LIN {X 0.001,Y -175.729,Z 1561.412,A 0.000,B 0.000,C 90.000,E1 254.212} C_DIS
LIN {X -0.003,Y -171.914,Z 1561.384,A 0.000,B 0.000,C 90.000,E1 249.082} C_DIS
LIN {X -0.028,Y -171.279,Z 1561.379,A 0.000,B 0.000,C 90.000,E1 248.230} C_DIS
LIN {X 0.018,Y -167.547,Z 1561.355,A 0.000,B 0.000,C 90.000,E1 243.896} C_DIS
LIN {X 0.032,Y -166.166,Z 1561.345,A 0.000,B 0.000,C 90.000,E1 242.153} C_DIS
LIN {X 0.022,Y -162.940,Z 1561.326,A 0.000,B 0.000,C 90.000,E1 238.663} C_DIS
LIN {X -0.001,Y -161.611,Z 1561.316,A 0.000,B 0.000,C 90.000,E1 236.914} C_DIS
LIN {X -0.025,Y -159.137,Z 1561.302,A 0.000,B 0.000,C 90.000,E1 234.276} C_DIS
LIN {X -0.014,Y -155.659,Z 1561.277,A 0.000,B 0.000,C 90.000,E1 229.828} C_DIS
LIN {X 0.038,Y -151.928,Z 1561.252,A 0.000,B 0.000,C 90.000,E1 225.324} C_DIS
LIN {X 0.053,Y -150.165,Z 1561.237,A 0.000,B 0.000,C 90.000,E1 222.609} C_DIS
LIN {X -0.027,Y -146.943,Z 1561.212,A 0.000,B 0.000,C 90.000,E1 218.096} C_DIS
LIN {X 0.079,Y -145.531,Z 1561.196,A 0.000,B 0.000,C 90.000,E1 215.311} C_DIS
LIN {X 0.000,Y -142.929,Z 1561.171,A 0.000,B 0.000,C 90.000,E1 210.747} C_DIS
LIN {X 0.000,Y -141.552,Z 1561.150,A 0.000,B 0.000,C 90.000,E1 207.052} C_DIS
LIN {X -0.011,Y -139.406,Z 1561.114,A 0.000,B 0.000,C 90.000,E1 200.556} C_DIS
LIN {X 0.042,Y -139.125,Z 1561.104,A 0.000,B 0.000,C 90.000,E1 198.671} C_DIS
LIN {X -0.063,Y -138.351,Z 1561.057,A 0.000,B 0.000,C 90.000,E1 190.310} C_DIS
LIN {X 0.064,Y -139.501,Z 1561.005,A 0.000,B 0.000,C 90.000,E1 180.917} C_DIS
LIN {X 0.005,Y -141.127,Z 1560.974,A 0.000,B 0.000,C 90.000,E1 175.355} C_DIS
LIN {X -0.041,Y -142.507,Z 1560.959,A 0.000,B 0.000,C 90.000,E1 172.591} C_DIS
LIN {X 0.045,Y -144.765,Z 1560.933,A 0.000,B 0.000,C 90.000,E1 167.937} C_DIS
LIN {X -0.005,Y -147.378,Z 1560.913,A 0.000,B 0.000,C 90.000,E1 164.283} C_DIS
LIN {X 0.058,Y -150.706,Z 1560.887,A 0.000,B 0.000,C 90.000,E1 159.699} C_DIS
LIN {X -0.001,Y -154.187,Z 1560.867,A 0.000,B 0.000,C 90.000,E1 156.102} C_DIS
LIN {X 0.068,Y -157.624,Z 1560.847,A 0.000,B 0.000,C 90.000,E1 152.487} C_DIS
LIN {X 0.017,Y -161.879,Z 1560.828,A 0.000,B 0.000,C 90.000,E1 148.948} C_DIS
LIN {X -0.011,Y -166.070,Z 1560.808,A 0.000,B 0.000,C 90.000,E1 145.435} C_DIS
LIN {X -0.010,Y -171.076,Z 1560.789,A 0.000,B 0.000,C 90.000,E1 141.949} C_DIS
LIN {X 0.045,Y -175.949,Z 1560.769,A 0.000,B 0.000,C 90.000,E1 138.485} C_DIS
LIN {X -0.095,Y -180.192,Z 1560.755,A 0.000,B 0.000,C 90.000,E1 135.972} C_DIS
LIN {X 0.010,Y -185.607,Z 1560.736,A 0.000,B 0.000,C 90.000,E1 132.567} C_DIS
LIN {X -0.078,Y -190.201,Z 1560.723,A 0.000,B 0.000,C 90.000,E1 130.092} C_DIS
LIN {X -0.034,Y -197.529,Z 1560.700,A 0.000,B 0.000,C 90.000,E1 125.964} C_DIS
LIN {X 0.007,Y -200.796,Z 1560.691,A 0.000,B 0.000,C 90.000,E1 124.326} C_DIS
LIN {X 0.030,Y -203.630,Z 1560.682,A 0.000,B 0.000,C 90.000,E1 122.704} C_DIS
LIN {X 0.011,Y -319.680,Z 1560.682,A 0.000,B 0.000,C 90.000,E1 122.704} C_DIS
LIN {X -0.131,Y -322.536,Z 1560.681,A 0.000,B 0.000,C 90.000,E1 122.673} C_DIS
LIN {X -0.011,Y -326.250,Z 1560.680,A 0.000,B 0.000,C 90.000,E1 122.467} C_DIS
LIN {X -0.066,Y -328.541,Z 1560.679,A 0.000,B 0.000,C 90.000,E1 122.291} C_DIS
LIN {X -0.102,Y -331.721,Z 1560.677,A 0.000,B 0.000,C 90.000,E1 121.926} C_DIS
LIN {X 0.040,Y -333.633,Z 1560.676,A 0.000,B 0.000,C 90.000,E1 121.592} C_DIS
LIN {X 0.184,Y -335.119,Z 1560.674,A 0.000,B 0.000,C 90.000,E1 121.258} C_DIS
LIN {X -0.201,Y -347.889,Z 1560.657,A 0.000,B 0.000,C 90.000,E1 118.231} C_DIS
LIN {X 0.062,Y -360.849,Z 1560.641,A 0.000,B 0.000,C 90.000,E1 115.463} C_DIS
LIN {X -0.104,Y -375.345,Z 1560.627,A 0.000,B 0.000,C 90.000,E1 112.823} C_DIS
LIN {X 0.048,Y -389.617,Z 1560.614,A 0.000,B 0.000,C 90.000,E1 110.482} C_DIS
LIN {X -0.079,Y -405.297,Z 1560.601,A 0.000,B 0.000,C 90.000,E1 108.236} C_DIS
LIN {X -0.073,Y -422.494,Z 1560.589,A 0.000,B 0.000,C 90.000,E1 106.024} C_DIS
LIN {X -0.171,Y -441.327,Z 1560.577,A 0.000,B 0.000,C 90.000,E1 103.883} C_DIS
LIN {X 0.024,Y -461.282,Z 1560.566,A 0.000,B 0.000,C 90.000,E1 101.827} C_DIS
LIN {X 0.129,Y -484.372,Z 1560.554,A 0.000,B 0.000,C 90.000,E1 99.726} C_DIS
LIN {X -0.075,Y -492.225,Z 1560.551,A 0.000,B 0.000,C 90.000,E1 99.095} C_DIS
LIN {X 0.121,Y -494.492,Z 1560.549,A 0.000,B 0.000,C 90.000,E1 98.859} C_DIS
LIN {X -0.171,Y -496.210,Z 1560.548,A 0.000,B 0.000,C 90.000,E1 98.681} C_DIS
LIN {X 0.161,Y -497.718,Z 1560.547,A 0.000,B 0.000,C 90.000,E1 98.398} C_DIS
LIN {X 0.076,Y -498.838,Z 1560.545,A 0.000,B 0.000,C 90.000,E1 98.163} C_DIS
LIN {X -0.149,Y -500.153,Z 1560.543,A 0.000,B 0.000,C 90.000,E1 97.701} C_DIS
LIN {X 0.129,Y -500.420,Z 1560.540,A 0.000,B 0.000,C 90.000,E1 97.182} C_DIS
LIN {X -0.082,Y -499.687,Z 1560.537,A 0.000,B 0.000,C 90.000,E1 96.720} C_DIS
LIN {X 0.206,Y -497.830,Z 1560.535,A 0.000,B 0.000,C 90.000,E1 96.201} C_DIS
LIN {X -0.007,Y -494.661,Z 1560.532,A 0.000,B 0.000,C 90.000,E1 95.739} C_DIS
LIN {X 0.042,Y -478.703,Z 1560.518,A 0.000,B 0.000,C 90.000,E1 93.269} C_DIS
LIN {X -0.049,Y -468.865,Z 1560.510,A 0.000,B 0.000,C 90.000,E1 91.776} C_DIS
LIN {X 0.123,Y -458.506,Z 1560.501,A 0.000,B 0.000,C 90.000,E1 90.229} C_DIS
LIN {X -0.099,Y -449.397,Z 1560.494,A 0.000,B 0.000,C 90.000,E1 88.969} C_DIS
LIN {X 0.015,Y -439.937,Z 1560.487,A 0.000,B 0.000,C 90.000,E1 87.650} C_DIS
LIN {X 0.131,Y -428.188,Z 1560.478,A 0.000,B 0.000,C 90.000,E1 86.045} C_DIS
LIN {X 0.189,Y -414.521,Z 1560.468,A 0.000,B 0.000,C 90.000,E1 84.147} C_DIS
LIN {X -0.172,Y -395.787,Z 1560.452,A 0.000,B 0.000,C 90.000,E1 81.432} C_DIS
LIN {X -0.071,Y -376.486,Z 1560.435,A 0.000,B 0.000,C 90.000,E1 78.285} C_DIS
LIN {X -0.026,Y -361.558,Z 1560.420,A 0.000,B 0.000,C 90.000,E1 75.644} C_DIS
LIN {X -0.138,Y -348.671,Z 1560.407,A 0.000,B 0.000,C 90.000,E1 73.268} C_DIS
LIN {X 0.078,Y -335.994,Z 1560.393,A 0.000,B 0.000,C 90.000,E1 70.786} C_DIS
LIN {X 0.056,Y -322.338,Z 1560.378,A 0.000,B 0.000,C 90.000,E1 67.975} C_DIS
LIN {X 0.048,Y -312.282,Z 1560.365,A 0.000,B 0.000,C 90.000,E1 65.741} C_DIS
LIN {X 0.103,Y -300.822,Z 1560.351,A 0.000,B 0.000,C 90.000,E1 63.127} C_DIS
LIN {X -0.098,Y -290.975,Z 1560.338,A 0.000,B 0.000,C 90.000,E1 60.845} C_DIS
LIN {X 0.028,Y -281.124,Z 1560.325,A 0.000,B 0.000,C 90.000,E1 58.456} C_DIS
LIN {X -0.135,Y -268.850,Z 1560.307,A 0.000,B 0.000,C 90.000,E1 55.388} C_DIS
LIN {X -0.076,Y -258.197,Z 1560.292,A 0.000,B 0.000,C 90.000,E1 52.557} C_DIS
LIN {X -0.003,Y -246.691,Z 1560.274,A 0.000,B 0.000,C 90.000,E1 49.299} C_DIS
LIN {X 0.047,Y -235.998,Z 1560.255,A 0.000,B 0.000,C 90.000,E1 45.972} C_DIS
LIN {X 0.018,Y -227.267,Z 1560.239,A 0.000,B 0.000,C 90.000,E1 42.975} C_DIS
LIN {X -0.017,Y -219.351,Z 1560.222,A 0.000,B 0.000,C 90.000,E1 39.930} C_DIS
LIN {X 0.120,Y -212.173,Z 1560.205,A 0.000,B 0.000,C 90.000,E1 36.790} C_DIS
LIN {X 0.045,Y -205.796,Z 1560.187,A 0.000,B 0.000,C 90.000,E1 33.658} C_DIS
LIN {X 0.048,Y -200.192,Z 1560.169,A 0.000,B 0.000,C 90.000,E1 30.463} C_DIS
LIN {X -0.046,Y -195.357,Z 1560.151,A 0.000,B 0.000,C 90.000,E1 27.257} C_DIS
LIN {X 0.003,Y -190.249,Z 1560.129,A 0.000,B 0.000,C 90.000,E1 23.153} C_DIS
LIN {X -0.042,Y -186.042,Z 1560.106,A 0.000,B 0.000,C 90.000,E1 19.033} C_DIS
LIN {X 0.003,Y -181.949,Z 1560.078,A 0.000,B 0.000,C 90.000,E1 14.008} C_DIS
LIN {X 0.022,Y -179.288,Z 1560.054,A 0.000,B 0.000,C 90.000,E1 9.792} C_DIS
LIN {X 0.074,Y -176.632,Z 1560.021,A 0.000,B 0.000,C 90.000,E1 3.841} C_DIS
LIN {X 0.076,Y -175.789,Z 1559.974,A 0.000,B 0.000,C 90.000,E1 355.241} C_DIS
LIN {X 0.028,Y -177.969,Z 1559.931,A 0.000,B 0.000,C 90.000,E1 347.589} C_DIS
LIN {X -0.093,Y -181.069,Z 1559.903,A 0.000,B 0.000,C 90.000,E1 342.543} C_DIS
LIN {X 0.078,Y -184.847,Z 1559.880,A 0.000,B 0.000,C 90.000,E1 338.284} C_DIS
LIN {X -0.043,Y -189.476,Z 1559.856,A 0.000,B 0.000,C 90.000,E1 334.152} C_DIS
LIN {X -0.028,Y -193.917,Z 1559.838,A 0.000,B 0.000,C 90.000,E1 330.845} C_DIS
LIN {X -0.049,Y -198.981,Z 1559.820,A 0.000,B 0.000,C 90.000,E1 327.582} C_DIS
LIN {X 0.046,Y -204.824,Z 1559.802,A 0.000,B 0.000,C 90.000,E1 324.322} C_DIS
LIN {X -0.094,Y -211.403,Z 1559.784,A 0.000,B 0.000,C 90.000,E1 321.170} C_DIS
LIN {X 0.001,Y -218.920,Z 1559.767,A 0.000,B 0.000,C 90.000,E1 318.000} C_DIS
LIN {X 0.062,Y -228.250,Z 1559.747,A 0.000,B 0.000,C 90.000,E1 314.514} C_DIS
LIN {X -0.049,Y -237.564,Z 1559.731,A 0.000,B 0.000,C 90.000,E1 311.515} C_DIS
LIN {X -0.017,Y -244.136,Z 1559.720,A 0.000,B 0.000,C 90.000,E1 309.644} C_DIS
LIN {X -0.035,Y -250.151,Z 1559.712,A 0.000,B 0.000,C 90.000,E1 308.177} C_DIS
LIN {X -0.103,Y -258.667,Z 1559.702,A 0.000,B 0.000,C 90.000,E1 306.377} C_DIS
LIN {X 0.121,Y -266.282,Z 1559.694,A 0.000,B 0.000,C 90.000,E1 304.898} C_DIS
LIN {X -0.001,Y -276.782,Z 1559.684,A 0.000,B 0.000,C 90.000,E1 303.166} C_DIS
LIN {X 0.063,Y -297.972,Z 1559.667,A 0.000,B 0.000,C 90.000,E1 300.079} C_DIS
LIN {X 0.067,Y -315.483,Z 1559.654,A 0.000,B 0.000,C 90.000,E1 297.769} C_DIS
LIN {X 0.063,Y -330.718,Z 1559.644,A 0.000,B 0.000,C 90.000,E1 295.848} C_DIS
LIN {X -0.091,Y -346.011,Z 1559.633,A 0.000,B 0.000,C 90.000,E1 294.003} C_DIS
LIN {X 0.134,Y -366.686,Z 1559.620,A 0.000,B 0.000,C 90.000,E1 291.589} C_DIS
LIN {X 0.107,Y -379.285,Z 1559.612,A 0.000,B 0.000,C 90.000,E1 290.194} C_DIS
LIN {X 0.153,Y -389.278,Z 1559.606,A 0.000,B 0.000,C 90.000,E1 289.033} C_DIS
LIN {X 0.119,Y -396.170,Z 1559.601,A 0.000,B 0.000,C 90.000,E1 288.181} C_DIS
LIN {X 0.032,Y -402.390,Z 1559.596,A 0.000,B 0.000,C 90.000,E1 287.347} C_DIS
LIN {X 0.114,Y -407.864,Z 1559.592,A 0.000,B 0.000,C 90.000,E1 286.496} C_DIS
LIN {X -0.086,Y -411.083,Z 1559.589,A 0.000,B 0.000,C 90.000,E1 285.969} C_DIS
LIN {X -0.036,Y -415.144,Z 1559.584,A 0.000,B 0.000,C 90.000,E1 285.134} C_DIS
LIN {X 0.046,Y -418.481,Z 1559.579,A 0.000,B 0.000,C 90.000,E1 284.300} C_DIS
LIN {X -0.084,Y -420.231,Z 1559.576,A 0.000,B 0.000,C 90.000,E1 283.772} C_DIS
LIN {X -0.111,Y -421.582,Z 1559.573,A 0.000,B 0.000,C 90.000,E1 283.231} C_DIS
LIN {X 0.184,Y -422.530,Z 1559.570,A 0.000,B 0.000,C 90.000,E1 282.647} C_DIS
LIN {X 0.076,Y -422.973,Z 1559.567,A 0.000,B 0.000,C 90.000,E1 282.119} C_DIS
LIN {X -0.025,Y -422.940,Z 1559.564,A 0.000,B 0.000,C 90.000,E1 281.591} C_DIS
LIN {X -0.207,Y -422.407,Z 1559.561,A 0.000,B 0.000,C 90.000,E1 281.074} C_DIS
LIN {X 0.108,Y -421.297,Z 1559.558,A 0.000,B 0.000,C 90.000,E1 280.489} C_DIS
LIN {X 0.005,Y -419.589,Z 1559.555,A 0.000,B 0.000,C 90.000,E1 279.962} C_DIS
LIN {X -0.107,Y -417.240,Z 1559.552,A 0.000,B 0.000,C 90.000,E1 279.434} C_DIS
LIN {X 0.107,Y -414.174,Z 1559.549,A 0.000,B 0.000,C 90.000,E1 278.859} C_DIS
LIN {X -0.101,Y -410.312,Z 1559.546,A 0.000,B 0.000,C 90.000,E1 278.341} C_DIS
LIN {X 0.137,Y -405.638,Z 1559.543,A 0.000,B 0.000,C 90.000,E1 277.757} C_DIS
LIN {X -0.110,Y -400.056,Z 1559.540,A 0.000,B 0.000,C 90.000,E1 277.239} C_DIS
LIN {X -0.046,Y -394.108,Z 1559.537,A 0.000,B 0.000,C 90.000,E1 276.720} C_DIS
LIN {X -0.043,Y -387.993,Z 1559.535,A 0.000,B 0.000,C 90.000,E1 276.258} C_DIS
LIN {X -0.145,Y -381.773,Z 1559.532,A 0.000,B 0.000,C 90.000,E1 275.853} C_DIS
LIN {X -0.039,Y -375.314,Z 1559.530,A 0.000,B 0.000,C 90.000,E1 275.454} C_DIS
LIN {X 0.086,Y -365.730,Z 1559.527,A 0.000,B 0.000,C 90.000,E1 274.935} C_DIS
LIN {X 0.155,Y -355.917,Z 1559.525,A 0.000,B 0.000,C 90.000,E1 274.473} C_DIS
LIN {X -0.030,Y -340.256,Z 1559.521,A 0.000,B 0.000,C 90.000,E1 273.841} C_DIS
LIN {X 0.136,Y -327.066,Z 1559.519,A 0.000,B 0.000,C 90.000,E1 273.326} C_DIS
LIN {X -0.086,Y -316.982,Z 1559.517,A 0.000,B 0.000,C 90.000,E1 273.037} C_DIS
LIN {X -0.084,Y -306.535,Z 1559.515,A 0.000,B 0.000,C 90.000,E1 272.751} C_DIS
LIN {X 0.118,Y -295.128,Z 1559.514,A 0.000,B 0.000,C 90.000,E1 272.465} C_DIS
LIN {X 0.004,Y -282.361,Z 1559.513,A 0.000,B 0.000,C 90.000,E1 272.293} C_DIS
LIN {X 0.048,Y -267.759,Z 1559.512,A 0.000,B 0.000,C 90.000,E1 272.121} C_DIS
LIN {X -0.013,Y -258.424,Z 1559.511,A 0.000,B 0.000,C 90.000,E1 272.064} C_DIS
LIN {X 0.060,Y -246.056,Z 1559.511,A 0.000,B 0.000,C 90.000,E1 272.007} C_DIS
LIN {X 0.016,Y -181.260,Z 1559.511,A 0.000,B 0.000,C 90.000,E1 272.007} C_DIS
LIN {X -0.008,Y -181.581,Z 1559.502,A 0.000,B 0.000,C 90.000,E1 270.286} C_DIS
LIN {X -0.032,Y -180.898,Z 1559.474,A 0.000,B 0.000,C 90.000,E1 265.241} C_DIS
LIN {X -0.083,Y -180.212,Z 1559.464,A 0.000,B 0.000,C 90.000,E1 263.571} C_DIS
LIN {X 0.047,Y -179.032,Z 1559.445,A 0.000,B 0.000,C 90.000,E1 260.151} C_DIS
LIN {X -0.066,Y -178.688,Z 1559.441,A 0.000,B 0.000,C 90.000,E1 259.342} C_DIS
LIN {X 0.044,Y -175.738,Z 1559.412,A 0.000,B 0.000,C 90.000,E1 254.212} C_DIS
LIN {X 0.040,Y -171.922,Z 1559.384,A 0.000,B 0.000,C 90.000,E1 249.082} C_DIS
LIN {X 0.014,Y -171.294,Z 1559.379,A 0.000,B 0.000,C 90.000,E1 248.230} C_DIS
LIN {X 0.060,Y -167.558,Z 1559.355,A 0.000,B 0.000,C 90.000,E1 243.896} C_DIS
LIN {X 0.074,Y -166.181,Z 1559.345,A 0.000,B 0.000,C 90.000,E1 242.153} C_DIS
LIN {X 0.063,Y -162.952,Z 1559.326,A 0.000,B 0.000,C 90.000,E1 238.663} C_DIS
LIN {X 0.111,Y -160.859,Z 1559.311,A 0.000,B 0.000,C 90.000,E1 236.008} C_DIS
LIN {X 0.088,Y -157.635,Z 1559.292,A 0.000,B 0.000,C 90.000,E1 232.477} C_DIS
LIN {X 0.025,Y -155.672,Z 1559.277,A 0.000,B 0.000,C 90.000,E1 229.828} C_DIS
LIN {X 0.077,Y -151.940,Z 1559.252,A 0.000,B 0.000,C 90.000,E1 225.324} C_DIS
LIN {X 0.092,Y -150.176,Z 1559.237,A 0.000,B 0.000,C 90.000,E1 222.609} C_DIS
LIN {X 0.012,Y -146.952,Z 1559.212,A 0.000,B 0.000,C 90.000,E1 218.096} C_DIS
LIN {X -0.001,Y -145.540,Z 1559.196,A 0.000,B 0.000,C 90.000,E1 215.358} C_DIS
LIN {X 0.039,Y -142.936,Z 1559.171,A 0.000,B 0.000,C 90.000,E1 210.747} C_DIS
LIN {X -0.027,Y -141.559,Z 1559.150,A 0.000,B 0.000,C 90.000,E1 207.078} C_DIS
LIN {X 0.026,Y -139.408,Z 1559.114,A 0.000,B 0.000,C 90.000,E1 200.556} C_DIS
LIN {X -0.053,Y -139.129,Z 1559.104,A 0.000,B 0.000,C 90.000,E1 198.725} C_DIS
LIN {X -0.025,Y -138.350,Z 1559.057,A 0.000,B 0.000,C 90.000,E1 190.310} C_DIS
LIN {X -0.037,Y -139.499,Z 1559.005,A 0.000,B 0.000,C 90.000,E1 180.974} C_DIS
LIN {X 0.044,Y -141.121,Z 1558.974,A 0.000,B 0.000,C 90.000,E1 175.355} C_DIS
LIN {X -0.004,Y -142.500,Z 1558.959,A 0.000,B 0.000,C 90.000,E1 172.591} C_DIS
LIN {X -0.057,Y -144.756,Z 1558.933,A 0.000,B 0.000,C 90.000,E1 167.993} C_DIS
LIN {X 0.034,Y -147.366,Z 1558.913,A 0.000,B 0.000,C 90.000,E1 164.283} C_DIS
LIN {X -0.043,Y -150.693,Z 1558.887,A 0.000,B 0.000,C 90.000,E1 159.752} C_DIS
LIN {X 0.039,Y -154.173,Z 1558.867,A 0.000,B 0.000,C 90.000,E1 156.102} C_DIS
LIN {X -0.031,Y -157.607,Z 1558.847,A 0.000,B 0.000,C 90.000,E1 152.538} C_DIS
LIN {X 0.058,Y -161.860,Z 1558.828,A 0.000,B 0.000,C 90.000,E1 148.948} C_DIS
LIN {X -0.063,Y -166.051,Z 1558.808,A 0.000,B 0.000,C 90.000,E1 145.468} C_DIS
LIN {X -0.072,Y -171.055,Z 1558.789,A 0.000,B 0.000,C 90.000,E1 141.984} C_DIS
LIN {X -0.043,Y -175.927,Z 1558.770,A 0.000,B 0.000,C 90.000,E1 138.528} C_DIS
LIN {X -0.051,Y -180.166,Z 1558.755,A 0.000,B 0.000,C 90.000,E1 135.972} C_DIS
LIN {X -0.082,Y -185.583,Z 1558.737,A 0.000,B 0.000,C 90.000,E1 132.609} C_DIS
LIN {X -0.033,Y -190.174,Z 1558.723,A 0.000,B 0.000,C 90.000,E1 130.092} C_DIS
LIN {X 0.012,Y -197.502,Z 1558.700,A 0.000,B 0.000,C 90.000,E1 125.964} C_DIS
LIN {X 0.054,Y -200.772,Z 1558.691,A 0.000,B 0.000,C 90.000,E1 124.326} C_DIS
LIN {X -0.015,Y -203.565,Z 1558.682,A 0.000,B 0.000,C 90.000,E1 122.752} C_DIS
LIN {X -0.066,Y -319.571,Z 1558.682,A 0.000,B 0.000,C 90.000,E1 122.752} C_DIS
LIN {X 0.011,Y -323.866,Z 1558.681,A 0.000,B 0.000,C 90.000,E1 122.625} C_DIS
LIN {X 0.047,Y -327.091,Z 1558.680,A 0.000,B 0.000,C 90.000,E1 122.418} C_DIS
LIN {X -0.010,Y -330.765,Z 1558.678,A 0.000,B 0.000,C 90.000,E1 122.054} C_DIS
LIN {X 0.142,Y -334.220,Z 1558.675,A 0.000,B 0.000,C 90.000,E1 121.465} C_DIS
LIN {X 0.026,Y -341.758,Z 1558.665,A 0.000,B 0.000,C 90.000,E1 119.617} C_DIS
LIN {X -0.029,Y -353.974,Z 1558.649,A 0.000,B 0.000,C 90.000,E1 116.873} C_DIS
LIN {X 0.103,Y -367.667,Z 1558.634,A 0.000,B 0.000,C 90.000,E1 114.155} C_DIS
LIN {X -0.132,Y -381.169,Z 1558.621,A 0.000,B 0.000,C 90.000,E1 111.844} C_DIS
LIN {X 0.040,Y -396.021,Z 1558.609,A 0.000,B 0.000,C 90.000,E1 109.523} C_DIS
LIN {X 0.078,Y -412.326,Z 1558.596,A 0.000,B 0.000,C 90.000,E1 107.275} C_DIS
LIN {X -0.260,Y -430.196,Z 1558.584,A 0.000,B 0.000,C 90.000,E1 105.134} C_DIS
LIN {X -0.186,Y -449.638,Z 1558.572,A 0.000,B 0.000,C 90.000,E1 103.008} C_DIS
LIN {X 0.139,Y -469.833,Z 1558.561,A 0.000,B 0.000,C 90.000,E1 101.007} C_DIS
LIN {X -0.190,Y -493.109,Z 1558.550,A 0.000,B 0.000,C 90.000,E1 99.029} C_DIS
LIN {X -0.082,Y -495.138,Z 1558.549,A 0.000,B 0.000,C 90.000,E1 98.803} C_DIS
LIN {X -0.171,Y -496.889,Z 1558.547,A 0.000,B 0.000,C 90.000,E1 98.568} C_DIS
LIN {X 0.233,Y -498.199,Z 1558.546,A 0.000,B 0.000,C 90.000,E1 98.276} C_DIS
LIN {X 0.002,Y -499.809,Z 1558.543,A 0.000,B 0.000,C 90.000,E1 97.814} C_DIS
LIN {X -0.221,Y -500.332,Z 1558.541,A 0.000,B 0.000,C 90.000,E1 97.352} C_DIS
LIN {X 0.062,Y -499.856,Z 1558.538,A 0.000,B 0.000,C 90.000,E1 96.834} C_DIS
LIN {X -0.148,Y -498.310,Z 1558.535,A 0.000,B 0.000,C 90.000,E1 96.372} C_DIS
LIN {X 0.214,Y -497.050,Z 1558.534,A 0.000,B 0.000,C 90.000,E1 96.087} C_DIS
LIN {X 0.193,Y -479.421,Z 1558.519,A 0.000,B 0.000,C 90.000,E1 93.383} C_DIS
LIN {X -0.190,Y -471.299,Z 1558.512,A 0.000,B 0.000,C 90.000,E1 92.178} C_DIS
LIN {X -0.212,Y -462.815,Z 1558.505,A 0.000,B 0.000,C 90.000,E1 90.917} C_DIS
LIN {X 0.087,Y -453.957,Z 1558.498,A 0.000,B 0.000,C 90.000,E1 89.599} C_DIS
LIN {X -0.193,Y -444.668,Z 1558.491,A 0.000,B 0.000,C 90.000,E1 88.339} C_DIS
LIN {X -0.154,Y -435.046,Z 1558.483,A 0.000,B 0.000,C 90.000,E1 87.020} C_DIS
LIN {X 0.060,Y -421.354,Z 1558.473,A 0.000,B 0.000,C 90.000,E1 85.122} C_DIS
LIN {X -0.143,Y -402.247,Z 1558.458,A 0.000,B 0.000,C 90.000,E1 82.413} C_DIS
LIN {X 0.058,Y -384.231,Z 1558.442,A 0.000,B 0.000,C 90.000,E1 79.567} C_DIS
LIN {X -0.126,Y -368.973,Z 1558.428,A 0.000,B 0.000,C 90.000,E1 76.992} C_DIS
LIN {X -0.141,Y -355.921,Z 1558.414,A 0.000,B 0.000,C 90.000,E1 74.629} C_DIS
LIN {X 0.037,Y -344.712,Z 1558.403,A 0.000,B 0.000,C 90.000,E1 72.489} C_DIS
LIN {X 0.127,Y -330.632,Z 1558.387,A 0.000,B 0.000,C 90.000,E1 69.699} C_DIS
LIN {X 0.062,Y -314.397,Z 1558.368,A 0.000,B 0.000,C 90.000,E1 66.230} C_DIS
LIN {X 0.008,Y -304.371,Z 1558.355,A 0.000,B 0.000,C 90.000,E1 63.973} C_DIS
LIN {X 0.140,Y -293.077,Z 1558.341,A 0.000,B 0.000,C 90.000,E1 61.307} C_DIS
LIN {X -0.081,Y -283.213,Z 1558.328,A 0.000,B 0.000,C 90.000,E1 58.997} C_DIS
LIN {X 0.105,Y -272.238,Z 1558.312,A 0.000,B 0.000,C 90.000,E1 56.215} C_DIS
LIN {X 0.142,Y -260.233,Z 1558.295,A 0.000,B 0.000,C 90.000,E1 53.050} C_DIS
LIN {X 0.110,Y -248.655,Z 1558.277,A 0.000,B 0.000,C 90.000,E1 49.828} C_DIS
LIN {X 0.046,Y -237.838,Z 1558.259,A 0.000,B 0.000,C 90.000,E1 46.539} C_DIS
LIN {X 0.013,Y -227.927,Z 1558.240,A 0.000,B 0.000,C 90.000,E1 43.176} C_DIS
LIN {X -0.021,Y -219.987,Z 1558.223,A 0.000,B 0.000,C 90.000,E1 40.135} C_DIS
LIN {X -0.001,Y -212.789,Z 1558.206,A 0.000,B 0.000,C 90.000,E1 37.030} C_DIS
LIN {X 0.065,Y -206.376,Z 1558.188,A 0.000,B 0.000,C 90.000,E1 33.865} C_DIS
LIN {X 0.083,Y -200.747,Z 1558.171,A 0.000,B 0.000,C 90.000,E1 30.669} C_DIS
LIN {X 0.004,Y -195.865,Z 1558.153,A 0.000,B 0.000,C 90.000,E1 27.462} C_DIS
LIN {X -0.025,Y -190.745,Z 1558.130,A 0.000,B 0.000,C 90.000,E1 23.387} C_DIS
LIN {X -0.062,Y -186.485,Z 1558.107,A 0.000,B 0.000,C 90.000,E1 19.268} C_DIS
LIN {X -0.005,Y -182.358,Z 1558.079,A 0.000,B 0.000,C 90.000,E1 14.245} C_DIS
LIN {X 0.060,Y -179.647,Z 1558.056,A 0.000,B 0.000,C 90.000,E1 10.018} C_DIS
LIN {X -0.072,Y -176.949,Z 1558.023,A 0.000,B 0.000,C 90.000,E1 4.131} C_DIS
LIN {X -0.091,Y -176.033,Z 1557.974,A 0.000,B 0.000,C 90.000,E1 355.298} C_DIS
LIN {X 0.049,Y -178.231,Z 1557.931,A 0.000,B 0.000,C 90.000,E1 347.589} C_DIS
LIN {X -0.061,Y -181.315,Z 1557.903,A 0.000,B 0.000,C 90.000,E1 342.543} C_DIS
LIN {X -0.054,Y -185.110,Z 1557.880,A 0.000,B 0.000,C 90.000,E1 338.337} C_DIS
LIN {X 0.006,Y -189.722,Z 1557.856,A 0.000,B 0.000,C 90.000,E1 334.152} C_DIS
LIN {X 0.029,Y -194.127,Z 1557.838,A 0.000,B 0.000,C 90.000,E1 330.845} C_DIS
LIN {X 0.014,Y -199.164,Z 1557.820,A 0.000,B 0.000,C 90.000,E1 327.582} C_DIS
LIN {X -0.004,Y -204.980,Z 1557.802,A 0.000,B 0.000,C 90.000,E1 324.356} C_DIS
LIN {X -0.018,Y -211.515,Z 1557.784,A 0.000,B 0.000,C 90.000,E1 321.170} C_DIS
LIN {X 0.082,Y -218.976,Z 1557.767,A 0.000,B 0.000,C 90.000,E1 318.000} C_DIS
LIN {X -0.022,Y -228.263,Z 1557.747,A 0.000,B 0.000,C 90.000,E1 314.555} C_DIS
LIN {X 0.033,Y -237.534,Z 1557.731,A 0.000,B 0.000,C 90.000,E1 311.515} C_DIS
LIN {X 0.068,Y -244.108,Z 1557.720,A 0.000,B 0.000,C 90.000,E1 309.644} C_DIS
LIN {X 0.051,Y -250.109,Z 1557.712,A 0.000,B 0.000,C 90.000,E1 308.177} C_DIS
LIN {X -0.015,Y -258.577,Z 1557.702,A 0.000,B 0.000,C 90.000,E1 306.377} C_DIS
LIN {X -0.110,Y -268.152,Z 1557.692,A 0.000,B 0.000,C 90.000,E1 304.612} C_DIS
LIN {X 0.028,Y -278.855,Z 1557.682,A 0.000,B 0.000,C 90.000,E1 302.832} C_DIS
LIN {X -0.102,Y -297.767,Z 1557.667,A 0.000,B 0.000,C 90.000,E1 300.129} C_DIS
LIN {X 0.160,Y -315.309,Z 1557.654,A 0.000,B 0.000,C 90.000,E1 297.769} C_DIS
LIN {X 0.158,Y -330.569,Z 1557.644,A 0.000,B 0.000,C 90.000,E1 295.848} C_DIS
LIN {X -0.078,Y -345.846,Z 1557.633,A 0.000,B 0.000,C 90.000,E1 294.027} C_DIS
LIN {X -0.063,Y -366.647,Z 1557.620,A 0.000,B 0.000,C 90.000,E1 291.642} C_DIS
LIN {X 0.219,Y -376.758,Z 1557.614,A 0.000,B 0.000,C 90.000,E1 290.482} C_DIS
LIN {X -0.216,Y -386.872,Z 1557.608,A 0.000,B 0.000,C 90.000,E1 289.396} C_DIS
LIN {X 0.105,Y -393.979,Z 1557.603,A 0.000,B 0.000,C 90.000,E1 288.489} C_DIS
LIN {X 0.112,Y -400.493,Z 1557.598,A 0.000,B 0.000,C 90.000,E1 287.638} C_DIS
LIN {X 0.065,Y -406.274,Z 1557.593,A 0.000,B 0.000,C 90.000,E1 286.804} C_DIS
LIN {X 0.066,Y -411.278,Z 1557.589,A 0.000,B 0.000,C 90.000,E1 285.969} C_DIS
LIN {X 0.119,Y -415.403,Z 1557.584,A 0.000,B 0.000,C 90.000,E1 285.134} C_DIS
LIN {X 0.205,Y -418.775,Z 1557.580,A 0.000,B 0.000,C 90.000,E1 284.300} C_DIS
LIN {X 0.077,Y -420.537,Z 1557.577,A 0.000,B 0.000,C 90.000,E1 283.772} C_DIS
LIN {X -0.045,Y -421.938,Z 1557.573,A 0.000,B 0.000,C 90.000,E1 283.244} C_DIS
LIN {X -0.063,Y -422.903,Z 1557.571,A 0.000,B 0.000,C 90.000,E1 282.703} C_DIS
LIN {X -0.169,Y -423.411,Z 1557.568,A 0.000,B 0.000,C 90.000,E1 282.175} C_DIS
LIN {X 0.144,Y -423.381,Z 1557.564,A 0.000,B 0.000,C 90.000,E1 281.591} C_DIS
LIN {X -0.035,Y -422.933,Z 1557.562,A 0.000,B 0.000,C 90.000,E1 281.074} C_DIS
LIN {X -0.131,Y -421.877,Z 1557.558,A 0.000,B 0.000,C 90.000,E1 280.546} C_DIS
LIN {X 0.182,Y -420.216,Z 1557.555,A 0.000,B 0.000,C 90.000,E1 279.962} C_DIS
LIN {X 0.004,Y -417.939,Z 1557.552,A 0.000,B 0.000,C 90.000,E1 279.443} C_DIS
LIN {X -0.121,Y -414.908,Z 1557.549,A 0.000,B 0.000,C 90.000,E1 278.916} C_DIS
LIN {X 0.085,Y -411.123,Z 1557.546,A 0.000,B 0.000,C 90.000,E1 278.341} C_DIS
LIN {X -0.078,Y -406.504,Z 1557.543,A 0.000,B 0.000,C 90.000,E1 277.814} C_DIS
LIN {X 0.080,Y -400.993,Z 1557.540,A 0.000,B 0.000,C 90.000,E1 277.239} C_DIS
LIN {X 0.135,Y -395.064,Z 1557.537,A 0.000,B 0.000,C 90.000,E1 276.720} C_DIS
LIN {X 0.170,Y -389.106,Z 1557.535,A 0.000,B 0.000,C 90.000,E1 276.258} C_DIS
LIN {X 0.036,Y -382.803,Z 1557.533,A 0.000,B 0.000,C 90.000,E1 275.853} C_DIS
LIN {X 0.134,Y -376.370,Z 1557.530,A 0.000,B 0.000,C 90.000,E1 275.454} C_DIS
LIN {X -0.145,Y -366.700,Z 1557.528,A 0.000,B 0.000,C 90.000,E1 274.992} C_DIS
LIN {X -0.060,Y -356.954,Z 1557.525,A 0.000,B 0.000,C 90.000,E1 274.531} C_DIS
LIN {X 0.090,Y -341.199,Z 1557.521,A 0.000,B 0.000,C 90.000,E1 273.841} C_DIS
LIN {X -0.066,Y -328.130,Z 1557.519,A 0.000,B 0.000,C 90.000,E1 273.383} C_DIS
LIN {X 0.051,Y -318.166,Z 1557.517,A 0.000,B 0.000,C 90.000,E1 273.037} C_DIS
LIN {X 0.034,Y -307.675,Z 1557.515,A 0.000,B 0.000,C 90.000,E1 272.751} C_DIS
LIN {X -0.062,Y -296.673,Z 1557.514,A 0.000,B 0.000,C 90.000,E1 272.522} C_DIS
LIN {X 0.106,Y -284.444,Z 1557.513,A 0.000,B 0.000,C 90.000,E1 272.293} C_DIS
LIN {X -0.127,Y -270.107,Z 1557.512,A 0.000,B 0.000,C 90.000,E1 272.178} C_DIS
LIN {X 0.074,Y -261.481,Z 1557.512,A 0.000,B 0.000,C 90.000,E1 272.064} C_DIS
LIN {X -0.118,Y -248.775,Z 1557.511,A 0.000,B 0.000,C 90.000,E1 272.064} C_DIS
LIN {X 0.065,Y -181.257,Z 1557.511,A 0.000,B 0.000,C 90.000,E1 272.007} C_DIS
LIN {X 0.023,Y -181.581,Z 1557.502,A 0.000,B 0.000,C 90.000,E1 270.286} C_DIS
LIN {X -0.002,Y -180.900,Z 1557.474,A 0.000,B 0.000,C 90.000,E1 265.241} C_DIS
LIN {X -0.052,Y -180.217,Z 1557.464,A 0.000,B 0.000,C 90.000,E1 263.571} C_DIS
LIN {X 0.077,Y -179.035,Z 1557.445,A 0.000,B 0.000,C 90.000,E1 260.151} C_DIS
LIN {X -0.036,Y -178.695,Z 1557.441,A 0.000,B 0.000,C 90.000,E1 259.342} C_DIS
LIN {X 0.075,Y -175.744,Z 1557.412,A 0.000,B 0.000,C 90.000,E1 254.212} C_DIS
LIN {X 0.070,Y -171.928,Z 1557.384,A 0.000,B 0.000,C 90.000,E1 249.082} C_DIS
LIN {X 0.044,Y -171.303,Z 1557.379,A 0.000,B 0.000,C 90.000,E1 248.230} C_DIS
LIN {X 0.089,Y -167.565,Z 1557.355,A 0.000,B 0.000,C 90.000,E1 243.896} C_DIS
LIN {X 0.103,Y -166.192,Z 1557.345,A 0.000,B 0.000,C 90.000,E1 242.153} C_DIS
LIN {X 0.091,Y -162.960,Z 1557.326,A 0.000,B 0.000,C 90.000,E1 238.663} C_DIS
LIN {X -0.084,Y -160.869,Z 1557.311,A 0.000,B 0.000,C 90.000,E1 236.087} C_DIS
LIN {X -0.106,Y -157.643,Z 1557.292,A 0.000,B 0.000,C 90.000,E1 232.557} C_DIS
LIN {X 0.054,Y -155.680,Z 1557.277,A 0.000,B 0.000,C 90.000,E1 229.828} C_DIS
LIN {X -0.002,Y -151.946,Z 1557.252,A 0.000,B 0.000,C 90.000,E1 225.364} C_DIS
LIN {X -0.093,Y -150.185,Z 1557.237,A 0.000,B 0.000,C 90.000,E1 222.690} C_DIS
LIN {X 0.039,Y -146.958,Z 1557.212,A 0.000,B 0.000,C 90.000,E1 218.096} C_DIS
LIN {X -0.058,Y -145.546,Z 1557.197,A 0.000,B 0.000,C 90.000,E1 215.391} C_DIS
LIN {X -0.058,Y -142.941,Z 1557.171,A 0.000,B 0.000,C 90.000,E1 210.797} C_DIS
LIN {X 0.000,Y -141.565,Z 1557.150,A 0.000,B 0.000,C 90.000,E1 207.078} C_DIS
LIN {X 0.052,Y -139.411,Z 1557.114,A 0.000,B 0.000,C 90.000,E1 200.556} C_DIS
LIN {X -0.026,Y -139.132,Z 1557.104,A 0.000,B 0.000,C 90.000,E1 198.725} C_DIS
LIN {X 0.001,Y -138.350,Z 1557.057,A 0.000,B 0.000,C 90.000,E1 190.310} C_DIS
LIN {X -0.011,Y -139.497,Z 1557.005,A 0.000,B 0.000,C 90.000,E1 180.974} C_DIS
LIN {X -0.071,Y -141.116,Z 1556.974,A 0.000,B 0.000,C 90.000,E1 175.412} C_DIS
LIN {X 0.023,Y -142.496,Z 1556.959,A 0.000,B 0.000,C 90.000,E1 172.591} C_DIS
LIN {X -0.030,Y -144.750,Z 1556.933,A 0.000,B 0.000,C 90.000,E1 167.993} C_DIS
LIN {X -0.081,Y -147.358,Z 1556.913,A 0.000,B 0.000,C 90.000,E1 164.338} C_DIS
LIN {X -0.017,Y -150.684,Z 1556.887,A 0.000,B 0.000,C 90.000,E1 159.752} C_DIS
LIN {X 0.067,Y -154.164,Z 1556.867,A 0.000,B 0.000,C 90.000,E1 156.102} C_DIS
LIN {X -0.002,Y -157.597,Z 1556.847,A 0.000,B 0.000,C 90.000,E1 152.538} C_DIS
LIN {X -0.052,Y -161.847,Z 1556.828,A 0.000,B 0.000,C 90.000,E1 148.997} C_DIS
LIN {X -0.034,Y -166.037,Z 1556.808,A 0.000,B 0.000,C 90.000,E1 145.468} C_DIS
LIN {X -0.043,Y -171.041,Z 1556.789,A 0.000,B 0.000,C 90.000,E1 141.984} C_DIS
LIN {X -0.013,Y -175.912,Z 1556.770,A 0.000,B 0.000,C 90.000,E1 138.528} C_DIS
LIN {X -0.020,Y -180.149,Z 1556.755,A 0.000,B 0.000,C 90.000,E1 135.972} C_DIS
LIN {X -0.051,Y -185.567,Z 1556.737,A 0.000,B 0.000,C 90.000,E1 132.609} C_DIS
LIN {X -0.001,Y -190.155,Z 1556.723,A 0.000,B 0.000,C 90.000,E1 130.092} C_DIS
LIN {X 0.018,Y -195.924,Z 1556.704,A 0.000,B 0.000,C 90.000,E1 126.790} C_DIS
LIN {X 0.087,Y -200.754,Z 1556.691,A 0.000,B 0.000,C 90.000,E1 124.326} C_DIS
LIN {X 0.100,Y -203.505,Z 1556.682,A 0.000,B 0.000,C 90.000,E1 122.752} C_DIS
LIN {X 0.123,Y -319.610,Z 1556.682,A 0.000,B 0.000,C 90.000,E1 122.752} C_DIS
LIN {X -0.096,Y -321.743,Z 1556.682,A 0.000,B 0.000,C 90.000,E1 122.752} C_DIS
LIN {X -0.164,Y -324.979,Z 1556.681,A 0.000,B 0.000,C 90.000,E1 122.625} C_DIS
LIN {X -0.061,Y -328.451,Z 1556.680,A 0.000,B 0.000,C 90.000,E1 122.339} C_DIS
LIN {X 0.001,Y -332.093,Z 1556.677,A 0.000,B 0.000,C 90.000,E1 121.878} C_DIS
LIN {X 0.114,Y -333.874,Z 1556.675,A 0.000,B 0.000,C 90.000,E1 121.544} C_DIS
LIN {X 0.072,Y -336.462,Z 1556.672,A 0.000,B 0.000,C 90.000,E1 120.924} C_DIS
LIN {X 0.023,Y -348.025,Z 1556.656,A 0.000,B 0.000,C 90.000,E1 118.153} C_DIS
LIN {X 0.135,Y -361.007,Z 1556.641,A 0.000,B 0.000,C 90.000,E1 115.412} C_DIS
LIN {X -0.017,Y -375.526,Z 1556.626,A 0.000,B 0.000,C 90.000,E1 112.770} C_DIS
LIN {X 0.150,Y -389.821,Z 1556.614,A 0.000,B 0.000,C 90.000,E1 110.429} C_DIS
LIN {X 0.037,Y -405.525,Z 1556.601,A 0.000,B 0.000,C 90.000,E1 108.181} C_DIS
LIN {X 0.060,Y -422.747,Z 1556.589,A 0.000,B 0.000,C 90.000,E1 105.969} C_DIS
LIN {X -0.022,Y -441.609,Z 1556.577,A 0.000,B 0.000,C 90.000,E1 103.828} C_DIS
LIN {X 0.205,Y -461.574,Z 1556.566,A 0.000,B 0.000,C 90.000,E1 101.771} C_DIS
LIN {X -0.132,Y -484.674,Z 1556.554,A 0.000,B 0.000,C 90.000,E1 99.726} C_DIS
LIN {X 0.231,Y -492.521,Z 1556.550,A 0.000,B 0.000,C 90.000,E1 99.029} C_DIS
LIN {X -0.163,Y -494.685,Z 1556.549,A 0.000,B 0.000,C 90.000,E1 98.859} C_DIS
LIN {X 0.007,Y -496.328,Z 1556.548,A 0.000,B 0.000,C 90.000,E1 98.624} C_DIS
LIN {X -0.151,Y -497.751,Z 1556.547,A 0.000,B 0.000,C 90.000,E1 98.398} C_DIS
LIN {X -0.236,Y -498.803,Z 1556.545,A 0.000,B 0.000,C 90.000,E1 98.163} C_DIS
LIN {X 0.034,Y -500.006,Z 1556.542,A 0.000,B 0.000,C 90.000,E1 97.644} C_DIS
LIN {X -0.184,Y -500.174,Z 1556.540,A 0.000,B 0.000,C 90.000,E1 97.182} C_DIS
LIN {X 0.101,Y -499.337,Z 1556.537,A 0.000,B 0.000,C 90.000,E1 96.663} C_DIS
LIN {X -0.108,Y -497.355,Z 1556.534,A 0.000,B 0.000,C 90.000,E1 96.201} C_DIS
LIN {X 0.057,Y -481.359,Z 1556.521,A 0.000,B 0.000,C 90.000,E1 93.726} C_DIS
LIN {X -0.010,Y -471.711,Z 1556.512,A 0.000,B 0.000,C 90.000,E1 92.236} C_DIS
LIN {X -0.034,Y -463.244,Z 1556.505,A 0.000,B 0.000,C 90.000,E1 90.974} C_DIS
LIN {X -0.181,Y -454.420,Z 1556.498,A 0.000,B 0.000,C 90.000,E1 89.714} C_DIS
LIN {X -0.009,Y -445.167,Z 1556.491,A 0.000,B 0.000,C 90.000,E1 88.396} C_DIS
LIN {X 0.038,Y -435.569,Z 1556.484,A 0.000,B 0.000,C 90.000,E1 87.078} C_DIS
LIN {X -0.203,Y -421.916,Z 1556.473,A 0.000,B 0.000,C 90.000,E1 85.241} C_DIS
LIN {X -0.040,Y -404.670,Z 1556.460,A 0.000,B 0.000,C 90.000,E1 82.761} C_DIS
LIN {X 0.157,Y -386.513,Z 1556.444,A 0.000,B 0.000,C 90.000,E1 79.926} C_DIS
LIN {X 0.018,Y -369.488,Z 1556.428,A 0.000,B 0.000,C 90.000,E1 77.061} C_DIS
LIN {X -0.001,Y -356.409,Z 1556.415,A 0.000,B 0.000,C 90.000,E1 74.700} C_DIS
LIN {X -0.140,Y -343.627,Z 1556.402,A 0.000,B 0.000,C 90.000,E1 72.308} C_DIS
LIN {X -0.072,Y -329.550,Z 1556.386,A 0.000,B 0.000,C 90.000,E1 69.518} C_DIS
LIN {X -0.166,Y -313.347,Z 1556.367,A 0.000,B 0.000,C 90.000,E1 66.049} C_DIS
LIN {X -0.105,Y -303.354,Z 1556.354,A 0.000,B 0.000,C 90.000,E1 63.768} C_DIS
LIN {X 0.012,Y -292.049,Z 1556.339,A 0.000,B 0.000,C 90.000,E1 61.101} C_DIS
LIN {X 0.018,Y -282.242,Z 1556.326,A 0.000,B 0.000,C 90.000,E1 58.742} C_DIS
LIN {X -0.055,Y -271.283,Z 1556.311,A 0.000,B 0.000,C 90.000,E1 56.008} C_DIS
LIN {X -0.091,Y -260.659,Z 1556.296,A 0.000,B 0.000,C 90.000,E1 53.210} C_DIS
LIN {X -0.128,Y -250.362,Z 1556.280,A 0.000,B 0.000,C 90.000,E1 50.356} C_DIS
LIN {X 0.042,Y -239.454,Z 1556.261,A 0.000,B 0.000,C 90.000,E1 47.025} C_DIS
LIN {X -0.122,Y -229.425,Z 1556.243,A 0.000,B 0.000,C 90.000,E1 43.704} C_DIS
LIN {X 0.051,Y -221.400,Z 1556.226,A 0.000,B 0.000,C 90.000,E1 40.620} C_DIS
LIN {X 0.072,Y -214.064,Z 1556.209,A 0.000,B 0.000,C 90.000,E1 37.523} C_DIS
LIN {X -0.005,Y -207.556,Z 1556.191,A 0.000,B 0.000,C 90.000,E1 34.405} C_DIS
LIN {X 0.043,Y -201.817,Z 1556.173,A 0.000,B 0.000,C 90.000,E1 31.209} C_DIS
LIN {X 0.087,Y -196.825,Z 1556.156,A 0.000,B 0.000,C 90.000,E1 27.975} C_DIS
LIN {X -0.089,Y -191.611,Z 1556.133,A 0.000,B 0.000,C 90.000,E1 23.951} C_DIS
LIN {X -0.030,Y -187.260,Z 1556.110,A 0.000,B 0.000,C 90.000,E1 19.812} C_DIS
LIN {X -0.075,Y -183.011,Z 1556.082,A 0.000,B 0.000,C 90.000,E1 14.828} C_DIS
LIN {X -0.065,Y -179.712,Z 1556.054,A 0.000,B 0.000,C 90.000,E1 9.782} C_DIS
LIN {X -0.024,Y -177.110,Z 1556.021,A 0.000,B 0.000,C 90.000,E1 3.841} C_DIS
LIN {X 0.065,Y -176.218,Z 1555.979,A 0.000,B 0.000,C 90.000,E1 356.102} C_DIS
LIN {X -0.012,Y -178.120,Z 1555.936,A 0.000,B 0.000,C 90.000,E1 348.465} C_DIS
LIN {X 0.003,Y -180.936,Z 1555.908,A 0.000,B 0.000,C 90.000,E1 343.378} C_DIS
LIN {X 0.048,Y -184.514,Z 1555.884,A 0.000,B 0.000,C 90.000,E1 339.156} C_DIS
LIN {X 0.085,Y -188.948,Z 1555.861,A 0.000,B 0.000,C 90.000,E1 334.973} C_DIS
LIN {X -0.011,Y -194.343,Z 1555.838,A 0.000,B 0.000,C 90.000,E1 330.873} C_DIS
LIN {X 0.078,Y -199.349,Z 1555.820,A 0.000,B 0.000,C 90.000,E1 327.582} C_DIS
LIN {X -0.101,Y -205.128,Z 1555.802,A 0.000,B 0.000,C 90.000,E1 324.402} C_DIS
LIN {X 0.057,Y -211.629,Z 1555.784,A 0.000,B 0.000,C 90.000,E1 321.170} C_DIS
LIN {X 0.016,Y -219.033,Z 1555.767,A 0.000,B 0.000,C 90.000,E1 318.038} C_DIS
LIN {X -0.097,Y -228.270,Z 1555.748,A 0.000,B 0.000,C 90.000,E1 314.595} C_DIS
LIN {X -0.035,Y -237.522,Z 1555.731,A 0.000,B 0.000,C 90.000,E1 311.553} C_DIS
LIN {X 0.020,Y -242.677,Z 1555.723,A 0.000,B 0.000,C 90.000,E1 310.048} C_DIS
LIN {X -0.052,Y -248.476,Z 1555.714,A 0.000,B 0.000,C 90.000,E1 308.588} C_DIS
LIN {X 0.050,Y -256.708,Z 1555.704,A 0.000,B 0.000,C 90.000,E1 306.744} C_DIS
LIN {X 0.037,Y -264.064,Z 1555.696,A 0.000,B 0.000,C 90.000,E1 305.311} C_DIS
LIN {X -0.117,Y -274.290,Z 1555.686,A 0.000,B 0.000,C 90.000,E1 303.579} C_DIS
LIN {X 0.047,Y -290.320,Z 1555.673,A 0.000,B 0.000,C 90.000,E1 301.131} C_DIS
LIN {X -0.056,Y -312.560,Z 1555.656,A 0.000,B 0.000,C 90.000,E1 298.153} C_DIS
LIN {X -0.123,Y -327.846,Z 1555.646,A 0.000,B 0.000,C 90.000,E1 296.232} C_DIS
LIN {X -0.037,Y -343.242,Z 1555.635,A 0.000,B 0.000,C 90.000,E1 294.335} C_DIS
LIN {X 0.210,Y -364.076,Z 1555.622,A 0.000,B 0.000,C 90.000,E1 291.897} C_DIS
LIN {X 0.092,Y -377.127,Z 1555.614,A 0.000,B 0.000,C 90.000,E1 290.482} C_DIS
LIN {X 0.115,Y -387.139,Z 1555.608,A 0.000,B 0.000,C 90.000,E1 289.341} C_DIS
LIN {X 0.071,Y -394.261,Z 1555.603,A 0.000,B 0.000,C 90.000,E1 288.489} C_DIS
LIN {X 0.081,Y -400.805,Z 1555.598,A 0.000,B 0.000,C 90.000,E1 287.638} C_DIS
LIN {X 0.035,Y -406.571,Z 1555.593,A 0.000,B 0.000,C 90.000,E1 286.804} C_DIS
LIN {X 0.040,Y -411.590,Z 1555.589,A 0.000,B 0.000,C 90.000,E1 285.969} C_DIS
LIN {X 0.096,Y -415.756,Z 1555.584,A 0.000,B 0.000,C 90.000,E1 285.134} C_DIS
LIN {X 0.185,Y -419.127,Z 1555.580,A 0.000,B 0.000,C 90.000,E1 284.300} C_DIS
LIN {X 0.058,Y -420.918,Z 1555.577,A 0.000,B 0.000,C 90.000,E1 283.772} C_DIS
LIN {X -0.061,Y -422.337,Z 1555.573,A 0.000,B 0.000,C 90.000,E1 283.244} C_DIS
LIN {X -0.078,Y -423.323,Z 1555.571,A 0.000,B 0.000,C 90.000,E1 282.703} C_DIS
LIN {X 0.234,Y -423.836,Z 1555.568,A 0.000,B 0.000,C 90.000,E1 282.119} C_DIS
LIN {X 0.136,Y -423.877,Z 1555.564,A 0.000,B 0.000,C 90.000,E1 281.591} C_DIS
LIN {X -0.042,Y -423.431,Z 1555.562,A 0.000,B 0.000,C 90.000,E1 281.074} C_DIS
LIN {X -0.135,Y -422.386,Z 1555.558,A 0.000,B 0.000,C 90.000,E1 280.546} C_DIS
LIN {X 0.181,Y -420.781,Z 1555.555,A 0.000,B 0.000,C 90.000,E1 279.962} C_DIS
LIN {X -0.079,Y -419.786,Z 1555.554,A 0.000,B 0.000,C 90.000,E1 279.726} C_DIS
LIN {X 0.006,Y -418.550,Z 1555.552,A 0.000,B 0.000,C 90.000,E1 279.443} C_DIS
LIN {X -0.116,Y -415.514,Z 1555.549,A 0.000,B 0.000,C 90.000,E1 278.916} C_DIS
LIN {X 0.093,Y -411.749,Z 1555.546,A 0.000,B 0.000,C 90.000,E1 278.341} C_DIS
LIN {X -0.189,Y -409.595,Z 1555.545,A 0.000,B 0.000,C 90.000,E1 278.106} C_DIS
LIN {X -0.011,Y -404.548,Z 1555.542,A 0.000,B 0.000,C 90.000,E1 277.530} C_DIS
LIN {X -0.046,Y -398.858,Z 1555.539,A 0.000,B 0.000,C 90.000,E1 277.004} C_DIS
LIN {X 0.200,Y -392.888,Z 1555.536,A 0.000,B 0.000,C 90.000,E1 276.486} C_DIS
LIN {X -0.020,Y -386.871,Z 1555.534,A 0.000,B 0.000,C 90.000,E1 276.087} C_DIS
LIN {X -0.082,Y -377.367,Z 1555.531,A 0.000,B 0.000,C 90.000,E1 275.511} C_DIS
LIN {X -0.006,Y -367.685,Z 1555.528,A 0.000,B 0.000,C 90.000,E1 274.992} C_DIS
LIN {X 0.085,Y -358.001,Z 1555.525,A 0.000,B 0.000,C 90.000,E1 274.531} C_DIS
LIN {X -0.020,Y -345.361,Z 1555.522,A 0.000,B 0.000,C 90.000,E1 274.012} C_DIS
LIN {X 0.094,Y -335.679,Z 1555.520,A 0.000,B 0.000,C 90.000,E1 273.612} C_DIS
LIN {X 0.026,Y -325.684,Z 1555.518,A 0.000,B 0.000,C 90.000,E1 273.269} C_DIS
LIN {X -0.108,Y -315.518,Z 1555.516,A 0.000,B 0.000,C 90.000,E1 272.980} C_DIS
LIN {X -0.042,Y -305.041,Z 1555.515,A 0.000,B 0.000,C 90.000,E1 272.694} C_DIS
LIN {X -0.039,Y -294.078,Z 1555.514,A 0.000,B 0.000,C 90.000,E1 272.465} C_DIS
LIN {X -0.130,Y -281.042,Z 1555.513,A 0.000,B 0.000,C 90.000,E1 272.293} C_DIS
LIN {X -0.040,Y -265.664,Z 1555.512,A 0.000,B 0.000,C 90.000,E1 272.121} C_DIS
LIN {X -0.041,Y -254.838,Z 1555.511,A 0.000,B 0.000,C 90.000,E1 272.064} C_DIS
LIN {X -0.085,Y -250.289,Z 1555.511,A 0.000,B 0.000,C 90.000,E1 272.064} C_DIS
LIN {X 0.088,Y -181.256,Z 1555.511,A 0.000,B 0.000,C 90.000,E1 272.007} C_DIS
LIN {X 0.042,Y -181.580,Z 1555.502,A 0.000,B 0.000,C 90.000,E1 270.286} C_DIS
LIN {X 0.017,Y -180.900,Z 1555.474,A 0.000,B 0.000,C 90.000,E1 265.241} C_DIS
LIN {X -0.033,Y -180.220,Z 1555.464,A 0.000,B 0.000,C 90.000,E1 263.571} C_DIS
LIN {X 0.096,Y -179.037,Z 1555.445,A 0.000,B 0.000,C 90.000,E1 260.151} C_DIS
LIN {X -0.018,Y -178.698,Z 1555.441,A 0.000,B 0.000,C 90.000,E1 259.342} C_DIS
LIN {X 0.093,Y -175.748,Z 1555.412,A 0.000,B 0.000,C 90.000,E1 254.212} C_DIS
LIN {X 0.087,Y -171.932,Z 1555.384,A 0.000,B 0.000,C 90.000,E1 249.082} C_DIS
LIN {X 0.062,Y -171.309,Z 1555.379,A 0.000,B 0.000,C 90.000,E1 248.230} C_DIS
LIN {X -0.043,Y -167.569,Z 1555.355,A 0.000,B 0.000,C 90.000,E1 243.948} C_DIS
LIN {X -0.104,Y -166.198,Z 1555.346,A 0.000,B 0.000,C 90.000,E1 242.231} C_DIS
LIN {X -0.029,Y -162.965,Z 1555.326,A 0.000,B 0.000,C 90.000,E1 238.712} C_DIS
LIN {X -0.067,Y -160.876,Z 1555.312,A 0.000,B 0.000,C 90.000,E1 236.087} C_DIS
LIN {X -0.088,Y -157.648,Z 1555.292,A 0.000,B 0.000,C 90.000,E1 232.557} C_DIS
LIN {X 0.071,Y -155.685,Z 1555.277,A 0.000,B 0.000,C 90.000,E1 229.828} C_DIS
LIN {X 0.015,Y -151.951,Z 1555.252,A 0.000,B 0.000,C 90.000,E1 225.364} C_DIS
LIN {X -0.076,Y -150.191,Z 1555.237,A 0.000,B 0.000,C 90.000,E1 222.690} C_DIS
LIN {X 0.055,Y -146.962,Z 1555.212,A 0.000,B 0.000,C 90.000,E1 218.096} C_DIS
LIN {X -0.041,Y -145.549,Z 1555.197,A 0.000,B 0.000,C 90.000,E1 215.391} C_DIS
LIN {X -0.042,Y -142.943,Z 1555.171,A 0.000,B 0.000,C 90.000,E1 210.797} C_DIS
LIN {X 0.016,Y -141.569,Z 1555.151,A 0.000,B 0.000,C 90.000,E1 207.078} C_DIS
LIN {X -0.063,Y -139.411,Z 1555.114,A 0.000,B 0.000,C 90.000,E1 200.610} C_DIS
LIN {X -0.010,Y -139.134,Z 1555.104,A 0.000,B 0.000,C 90.000,E1 198.725} C_DIS
LIN {X 0.016,Y -138.350,Z 1555.057,A 0.000,B 0.000,C 90.000,E1 190.310} C_DIS
LIN {X 0.005,Y -139.495,Z 1555.005,A 0.000,B 0.000,C 90.000,E1 180.974} C_DIS
LIN {X -0.055,Y -141.114,Z 1554.974,A 0.000,B 0.000,C 90.000,E1 175.412} C_DIS
LIN {X 0.039,Y -142.493,Z 1554.959,A 0.000,B 0.000,C 90.000,E1 172.591} C_DIS
LIN {X -0.013,Y -144.745,Z 1554.933,A 0.000,B 0.000,C 90.000,E1 167.993} C_DIS
LIN {X -0.063,Y -147.353,Z 1554.913,A 0.000,B 0.000,C 90.000,E1 164.338} C_DIS
LIN {X 0.000,Y -150.679,Z 1554.888,A 0.000,B 0.000,C 90.000,E1 159.752} C_DIS
LIN {X 0.084,Y -154.158,Z 1554.867,A 0.000,B 0.000,C 90.000,E1 156.102} C_DIS
LIN {X 0.015,Y -157.590,Z 1554.847,A 0.000,B 0.000,C 90.000,E1 152.538} C_DIS
LIN {X -0.034,Y -161.839,Z 1554.828,A 0.000,B 0.000,C 90.000,E1 148.997} C_DIS
LIN {X -0.016,Y -166.029,Z 1554.808,A 0.000,B 0.000,C 90.000,E1 145.468} C_DIS
LIN {X -0.025,Y -171.032,Z 1554.789,A 0.000,B 0.000,C 90.000,E1 141.984} C_DIS
LIN {X 0.006,Y -175.903,Z 1554.770,A 0.000,B 0.000,C 90.000,E1 138.528} C_DIS
LIN {X 0.010,Y -181.506,Z 1554.751,A 0.000,B 0.000,C 90.000,E1 135.121} C_DIS
LIN {X 0.017,Y -187.025,Z 1554.732,A 0.000,B 0.000,C 90.000,E1 131.757} C_DIS
LIN {X 0.018,Y -190.144,Z 1554.723,A 0.000,B 0.000,C 90.000,E1 130.092} C_DIS
LIN {X 0.037,Y -195.913,Z 1554.704,A 0.000,B 0.000,C 90.000,E1 126.790} C_DIS
LIN {X 0.107,Y -200.744,Z 1554.691,A 0.000,B 0.000,C 90.000,E1 124.326} C_DIS
LIN {X -0.062,Y -203.444,Z 1554.682,A 0.000,B 0.000,C 90.000,E1 122.832} C_DIS
LIN {X -0.132,Y -319.477,Z 1554.682,A 0.000,B 0.000,C 90.000,E1 122.832} C_DIS
LIN {X -0.065,Y -322.470,Z 1554.682,A 0.000,B 0.000,C 90.000,E1 122.752} C_DIS
LIN {X 0.198,Y -325.622,Z 1554.681,A 0.000,B 0.000,C 90.000,E1 122.546} C_DIS
LIN {X 0.043,Y -329.223,Z 1554.679,A 0.000,B 0.000,C 90.000,E1 122.260} C_DIS
LIN {X -0.167,Y -332.802,Z 1554.677,A 0.000,B 0.000,C 90.000,E1 121.799} C_DIS
LIN {X -0.051,Y -334.389,Z 1554.675,A 0.000,B 0.000,C 90.000,E1 121.465} C_DIS
LIN {X 0.166,Y -348.470,Z 1554.656,A 0.000,B 0.000,C 90.000,E1 118.025} C_DIS
LIN {X -0.029,Y -361.508,Z 1554.641,A 0.000,B 0.000,C 90.000,E1 115.335} C_DIS
LIN {X 0.165,Y -376.087,Z 1554.626,A 0.000,B 0.000,C 90.000,E1 112.642} C_DIS
LIN {X -0.016,Y -390.439,Z 1554.613,A 0.000,B 0.000,C 90.000,E1 110.355} C_DIS
LIN {X -0.130,Y -406.205,Z 1554.600,A 0.000,B 0.000,C 90.000,E1 108.109} C_DIS
LIN {X -0.108,Y -423.495,Z 1554.588,A 0.000,B 0.000,C 90.000,E1 105.898} C_DIS
LIN {X 0.134,Y -442.430,Z 1554.576,A 0.000,B 0.000,C 90.000,E1 103.716} C_DIS
LIN {X -0.018,Y -462.420,Z 1554.565,A 0.000,B 0.000,C 90.000,E1 101.715} C_DIS
LIN {X 0.178,Y -485.546,Z 1554.553,A 0.000,B 0.000,C 90.000,E1 99.613} C_DIS
LIN {X 0.079,Y -493.297,Z 1554.550,A 0.000,B 0.000,C 90.000,E1 98.973} C_DIS
LIN {X 0.132,Y -495.279,Z 1554.549,A 0.000,B 0.000,C 90.000,E1 98.746} C_DIS
LIN {X -0.231,Y -496.794,Z 1554.547,A 0.000,B 0.000,C 90.000,E1 98.568} C_DIS
LIN {X 0.178,Y -498.070,Z 1554.546,A 0.000,B 0.000,C 90.000,E1 98.276} C_DIS
LIN {X 0.022,Y -499.002,Z 1554.545,A 0.000,B 0.000,C 90.000,E1 98.049} C_DIS
LIN {X -0.200,Y -500.006,Z 1554.542,A 0.000,B 0.000,C 90.000,E1 97.587} C_DIS
LIN {X 0.081,Y -499.993,Z 1554.539,A 0.000,B 0.000,C 90.000,E1 97.068} C_DIS
LIN {X -0.130,Y -498.964,Z 1554.537,A 0.000,B 0.000,C 90.000,E1 96.606} C_DIS
LIN {X -0.207,Y -498.022,Z 1554.535,A 0.000,B 0.000,C 90.000,E1 96.372} C_DIS
LIN {X 0.156,Y -496.735,Z 1554.534,A 0.000,B 0.000,C 90.000,E1 96.087} C_DIS
LIN {X 0.123,Y -479.110,Z 1554.519,A 0.000,B 0.000,C 90.000,E1 93.383} C_DIS
LIN {X 0.211,Y -471.021,Z 1554.512,A 0.000,B 0.000,C 90.000,E1 92.121} C_DIS
LIN {X 0.174,Y -462.524,Z 1554.505,A 0.000,B 0.000,C 90.000,E1 90.859} C_DIS
LIN {X 0.013,Y -453.682,Z 1554.498,A 0.000,B 0.000,C 90.000,E1 89.599} C_DIS
LIN {X -0.065,Y -442.554,Z 1554.489,A 0.000,B 0.000,C 90.000,E1 88.051} C_DIS
LIN {X 0.105,Y -430.937,Z 1554.480,A 0.000,B 0.000,C 90.000,E1 86.445} C_DIS
LIN {X 0.188,Y -417.325,Z 1554.470,A 0.000,B 0.000,C 90.000,E1 84.552} C_DIS
LIN {X -0.185,Y -400.276,Z 1554.456,A 0.000,B 0.000,C 90.000,E1 82.129} C_DIS
LIN {X -0.053,Y -382.397,Z 1554.440,A 0.000,B 0.000,C 90.000,E1 79.285} C_DIS
LIN {X 0.145,Y -367.245,Z 1554.426,A 0.000,B 0.000,C 90.000,E1 76.645} C_DIS
LIN {X 0.072,Y -354.255,Z 1554.413,A 0.000,B 0.000,C 90.000,E1 74.283} C_DIS
LIN {X -0.025,Y -343.092,Z 1554.401,A 0.000,B 0.000,C 90.000,E1 72.181} C_DIS
LIN {X 0.027,Y -328.991,Z 1554.385,A 0.000,B 0.000,C 90.000,E1 69.390} C_DIS
LIN {X -0.087,Y -312.782,Z 1554.366,A 0.000,B 0.000,C 90.000,E1 65.921} C_DIS
LIN {X -0.039,Y -302.819,Z 1554.354,A 0.000,B 0.000,C 90.000,E1 63.640} C_DIS
LIN {X 0.062,Y -291.556,Z 1554.339,A 0.000,B 0.000,C 90.000,E1 60.973} C_DIS
LIN {X 0.018,Y -280.359,Z 1554.324,A 0.000,B 0.000,C 90.000,E1 58.280} C_DIS
LIN {X 0.048,Y -269.471,Z 1554.308,A 0.000,B 0.000,C 90.000,E1 55.515} C_DIS
LIN {X -0.037,Y -258.940,Z 1554.293,A 0.000,B 0.000,C 90.000,E1 52.718} C_DIS
LIN {X 0.055,Y -247.521,Z 1554.275,A 0.000,B 0.000,C 90.000,E1 49.461} C_DIS
LIN {X 0.121,Y -236.840,Z 1554.256,A 0.000,B 0.000,C 90.000,E1 46.134} C_DIS
LIN {X 0.065,Y -227.114,Z 1554.238,A 0.000,B 0.000,C 90.000,E1 42.771} C_DIS
LIN {X 0.032,Y -219.324,Z 1554.221,A 0.000,B 0.000,C 90.000,E1 39.725} C_DIS
LIN {X -0.001,Y -212.263,Z 1554.203,A 0.000,B 0.000,C 90.000,E1 36.629} C_DIS
LIN {X -0.075,Y -205.997,Z 1554.186,A 0.000,B 0.000,C 90.000,E1 33.499} C_DIS
LIN {X 0.102,Y -200.501,Z 1554.168,A 0.000,B 0.000,C 90.000,E1 30.256} C_DIS
LIN {X 0.011,Y -195.757,Z 1554.150,A 0.000,B 0.000,C 90.000,E1 27.052} C_DIS
LIN {X 0.065,Y -190.798,Z 1554.128,A 0.000,B 0.000,C 90.000,E1 22.950} C_DIS
LIN {X -0.036,Y -186.608,Z 1554.105,A 0.000,B 0.000,C 90.000,E1 18.852} C_DIS
LIN {X 0.027,Y -182.539,Z 1554.077,A 0.000,B 0.000,C 90.000,E1 13.828} C_DIS
LIN {X -0.046,Y -179.402,Z 1554.049,A 0.000,B 0.000,C 90.000,E1 8.803} C_DIS
LIN {X 0.000,Y -176.939,Z 1554.011,A 0.000,B 0.000,C 90.000,E1 2.007} C_DIS
LIN {X -0.081,Y -177.179,Z 1553.955,A 0.000,B 0.000,C 90.000,E1 351.894} C_DIS
LIN {X -0.035,Y -179.621,Z 1553.922,A 0.000,B 0.000,C 90.000,E1 345.936} C_DIS
LIN {X 0.034,Y -182.497,Z 1553.898,A 0.000,B 0.000,C 90.000,E1 341.692} C_DIS
LIN {X 0.079,Y -186.397,Z 1553.875,A 0.000,B 0.000,C 90.000,E1 337.486} C_DIS
LIN {X -0.090,Y -191.230,Z 1553.852,A 0.000,B 0.000,C 90.000,E1 333.384} C_DIS
LIN {X -0.035,Y -195.740,Z 1553.834,A 0.000,B 0.000,C 90.000,E1 330.078} C_DIS
LIN {X -0.081,Y -200.896,Z 1553.816,A 0.000,B 0.000,C 90.000,E1 326.834} C_DIS
LIN {X 0.057,Y -206.842,Z 1553.798,A 0.000,B 0.000,C 90.000,E1 323.577} C_DIS
LIN {X -0.076,Y -213.496,Z 1553.780,A 0.000,B 0.000,C 90.000,E1 320.436} C_DIS
LIN {X -0.026,Y -222.065,Z 1553.760,A 0.000,B 0.000,C 90.000,E1 316.905} C_DIS
LIN {X -0.142,Y -230.494,Z 1553.744,A 0.000,B 0.000,C 90.000,E1 313.866} C_DIS
LIN {X -0.028,Y -239.995,Z 1553.727,A 0.000,B 0.000,C 90.000,E1 310.825} C_DIS
LIN {X 0.043,Y -246.915,Z 1553.716,A 0.000,B 0.000,C 90.000,E1 308.955} C_DIS
LIN {X -0.079,Y -254.888,Z 1553.706,A 0.000,B 0.000,C 90.000,E1 307.156} C_DIS
LIN {X 0.134,Y -263.946,Z 1553.696,A 0.000,B 0.000,C 90.000,E1 305.311} C_DIS
LIN {X 0.059,Y -272.015,Z 1553.688,A 0.000,B 0.000,C 90.000,E1 303.913} C_DIS
LIN {X -0.124,Y -283.067,Z 1553.679,A 0.000,B 0.000,C 90.000,E1 302.212} C_DIS
LIN {X 0.102,Y -302.259,Z 1553.664,A 0.000,B 0.000,C 90.000,E1 299.461} C_DIS
LIN {X -0.007,Y -317.476,Z 1553.653,A 0.000,B 0.000,C 90.000,E1 297.513} C_DIS
LIN {X 0.043,Y -332.759,Z 1553.642,A 0.000,B 0.000,C 90.000,E1 295.591} C_DIS
LIN {X -0.119,Y -348.206,Z 1553.632,A 0.000,B 0.000,C 90.000,E1 293.770} C_DIS
LIN {X 0.008,Y -369.027,Z 1553.619,A 0.000,B 0.000,C 90.000,E1 291.408} C_DIS
LIN {X -0.171,Y -379.328,Z 1553.613,A 0.000,B 0.000,C 90.000,E1 290.301} C_DIS
LIN {X 0.109,Y -386.938,Z 1553.608,A 0.000,B 0.000,C 90.000,E1 289.396} C_DIS
LIN {X 0.060,Y -394.094,Z 1553.603,A 0.000,B 0.000,C 90.000,E1 288.544} C_DIS
LIN {X 0.068,Y -400.675,Z 1553.598,A 0.000,B 0.000,C 90.000,E1 287.692} C_DIS
LIN {X 0.019,Y -406.488,Z 1553.594,A 0.000,B 0.000,C 90.000,E1 286.858} C_DIS
LIN {X -0.077,Y -409.993,Z 1553.591,A 0.000,B 0.000,C 90.000,E1 286.315} C_DIS
LIN {X -0.046,Y -414.500,Z 1553.586,A 0.000,B 0.000,C 90.000,E1 285.481} C_DIS
LIN {X -0.075,Y -418.165,Z 1553.581,A 0.000,B 0.000,C 90.000,E1 284.662} C_DIS
LIN {X 0.035,Y -421.101,Z 1553.577,A 0.000,B 0.000,C 90.000,E1 283.828} C_DIS
LIN {X -0.085,Y -422.581,Z 1553.574,A 0.000,B 0.000,C 90.000,E1 283.300} C_DIS
LIN {X -0.194,Y -423.656,Z 1553.571,A 0.000,B 0.000,C 90.000,E1 282.771} C_DIS
LIN {X 0.121,Y -424.224,Z 1553.568,A 0.000,B 0.000,C 90.000,E1 282.187} C_DIS
LIN {X 0.028,Y -424.382,Z 1553.565,A 0.000,B 0.000,C 90.000,E1 281.658} C_DIS
LIN {X -0.062,Y -423.962,Z 1553.562,A 0.000,B 0.000,C 90.000,E1 281.130} C_DIS
LIN {X -0.154,Y -423.085,Z 1553.559,A 0.000,B 0.000,C 90.000,E1 280.602} C_DIS
LIN {X 0.167,Y -421.552,Z 1553.556,A 0.000,B 0.000,C 90.000,E1 280.018} C_DIS
LIN {X -0.007,Y -419.405,Z 1553.553,A 0.000,B 0.000,C 90.000,E1 279.500} C_DIS
LIN {X -0.118,Y -416.507,Z 1553.550,A 0.000,B 0.000,C 90.000,E1 278.973} C_DIS
LIN {X 0.097,Y -412.809,Z 1553.547,A 0.000,B 0.000,C 90.000,E1 278.398} C_DIS
LIN {X -0.058,Y -408.351,Z 1553.544,A 0.000,B 0.000,C 90.000,E1 277.871} C_DIS
LIN {X 0.110,Y -402.957,Z 1553.541,A 0.000,B 0.000,C 90.000,E1 277.296} C_DIS
LIN {X 0.137,Y -397.102,Z 1553.538,A 0.000,B 0.000,C 90.000,E1 276.777} C_DIS
LIN {X 0.120,Y -391.053,Z 1553.535,A 0.000,B 0.000,C 90.000,E1 276.315} C_DIS
LIN {X 0.020,Y -384.882,Z 1553.533,A 0.000,B 0.000,C 90.000,E1 275.910} C_DIS
LIN {X 0.156,Y -378.648,Z 1553.531,A 0.000,B 0.000,C 90.000,E1 275.511} C_DIS
LIN {X -0.183,Y -368.822,Z 1553.528,A 0.000,B 0.000,C 90.000,E1 275.049} C_DIS
LIN {X -0.073,Y -359.213,Z 1553.525,A 0.000,B 0.000,C 90.000,E1 274.588} C_DIS
LIN {X 0.155,Y -346.571,Z 1553.522,A 0.000,B 0.000,C 90.000,E1 274.012} C_DIS
LIN {X -0.077,Y -336.856,Z 1553.520,A 0.000,B 0.000,C 90.000,E1 273.669} C_DIS
LIN {X -0.108,Y -327.137,Z 1553.518,A 0.000,B 0.000,C 90.000,E1 273.326} C_DIS
LIN {X 0.050,Y -316.877,Z 1553.517,A 0.000,B 0.000,C 90.000,E1 272.980} C_DIS
LIN {X 0.104,Y -306.445,Z 1553.515,A 0.000,B 0.000,C 90.000,E1 272.694} C_DIS
LIN {X 0.083,Y -295.749,Z 1553.514,A 0.000,B 0.000,C 90.000,E1 272.465} C_DIS
LIN {X -0.045,Y -282.969,Z 1553.513,A 0.000,B 0.000,C 90.000,E1 272.293} C_DIS
LIN {X 0.029,Y -267.674,Z 1553.512,A 0.000,B 0.000,C 90.000,E1 272.121} C_DIS
LIN {X -0.029,Y -254.704,Z 1553.511,A 0.000,B 0.000,C 90.000,E1 272.064} C_DIS
LIN {X -0.074,Y -247.980,Z 1553.511,A 0.000,B 0.000,C 90.000,E1 272.064} C_DIS
LIN {X -0.088,Y -181.255,Z 1553.511,A 0.000,B 0.000,C 90.000,E1 272.064} C_DIS
LIN {X 0.072,Y -181.581,Z 1553.502,A 0.000,B 0.000,C 90.000,E1 270.286} C_DIS
LIN {X 0.047,Y -180.901,Z 1553.474,A 0.000,B 0.000,C 90.000,E1 265.241} C_DIS
LIN {X -0.004,Y -180.225,Z 1553.464,A 0.000,B 0.000,C 90.000,E1 263.571} C_DIS
LIN {X -0.051,Y -179.039,Z 1553.446,A 0.000,B 0.000,C 90.000,E1 260.208} C_DIS
LIN {X 0.012,Y -178.705,Z 1553.441,A 0.000,B 0.000,C 90.000,E1 259.342} C_DIS
LIN {X -0.047,Y -175.753,Z 1553.412,A 0.000,B 0.000,C 90.000,E1 254.267} C_DIS
LIN {X -0.045,Y -171.937,Z 1553.384,A 0.000,B 0.000,C 90.000,E1 249.135} C_DIS
LIN {X -0.068,Y -171.318,Z 1553.379,A 0.000,B 0.000,C 90.000,E1 248.284} C_DIS
LIN {X -0.014,Y -167.576,Z 1553.355,A 0.000,B 0.000,C 90.000,E1 243.948} C_DIS
LIN {X -0.075,Y -166.208,Z 1553.346,A 0.000,B 0.000,C 90.000,E1 242.231} C_DIS
LIN {X -0.087,Y -162.973,Z 1553.326,A 0.000,B 0.000,C 90.000,E1 238.742} C_DIS
LIN {X -0.039,Y -160.886,Z 1553.312,A 0.000,B 0.000,C 90.000,E1 236.087} C_DIS
LIN {X -0.060,Y -157.656,Z 1553.292,A 0.000,B 0.000,C 90.000,E1 232.557} C_DIS
LIN {X -0.003,Y -155.694,Z 1553.277,A 0.000,B 0.000,C 90.000,E1 229.865} C_DIS
LIN {X -0.066,Y -151.958,Z 1553.252,A 0.000,B 0.000,C 90.000,E1 225.405} C_DIS
LIN {X -0.050,Y -150.199,Z 1553.237,A 0.000,B 0.000,C 90.000,E1 222.690} C_DIS
LIN {X 0.082,Y -146.968,Z 1553.212,A 0.000,B 0.000,C 90.000,E1 218.096} C_DIS
LIN {X -0.016,Y -145.555,Z 1553.197,A 0.000,B 0.000,C 90.000,E1 215.391} C_DIS
LIN {X -0.016,Y -142.948,Z 1553.171,A 0.000,B 0.000,C 90.000,E1 210.797} C_DIS
LIN {X 0.041,Y -141.574,Z 1553.151,A 0.000,B 0.000,C 90.000,E1 207.078} C_DIS
LIN {X -0.037,Y -139.413,Z 1553.114,A 0.000,B 0.000,C 90.000,E1 200.610} C_DIS
LIN {X 0.016,Y -139.136,Z 1553.104,A 0.000,B 0.000,C 90.000,E1 198.725} C_DIS
LIN {X 0.042,Y -138.348,Z 1553.057,A 0.000,B 0.000,C 90.000,E1 190.310} C_DIS
LIN {X 0.030,Y -139.494,Z 1553.005,A 0.000,B 0.000,C 90.000,E1 180.974} C_DIS
LIN {X -0.030,Y -141.108,Z 1552.974,A 0.000,B 0.000,C 90.000,E1 175.412} C_DIS
LIN {X 0.065,Y -142.488,Z 1552.959,A 0.000,B 0.000,C 90.000,E1 172.591} C_DIS
LIN {X 0.012,Y -144.739,Z 1552.933,A 0.000,B 0.000,C 90.000,E1 167.993} C_DIS
LIN {X -0.038,Y -147.345,Z 1552.913,A 0.000,B 0.000,C 90.000,E1 164.338} C_DIS
LIN {X 0.027,Y -150.670,Z 1552.888,A 0.000,B 0.000,C 90.000,E1 159.752} C_DIS
LIN {X -0.092,Y -154.149,Z 1552.867,A 0.000,B 0.000,C 90.000,E1 156.177} C_DIS
LIN {X 0.043,Y -157.579,Z 1552.848,A 0.000,B 0.000,C 90.000,E1 152.538} C_DIS
LIN {X -0.006,Y -161.826,Z 1552.828,A 0.000,B 0.000,C 90.000,E1 148.997} C_DIS
LIN {X 0.013,Y -166.016,Z 1552.808,A 0.000,B 0.000,C 90.000,E1 145.468} C_DIS
LIN {X 0.004,Y -171.017,Z 1552.789,A 0.000,B 0.000,C 90.000,E1 141.984} C_DIS
LIN {X 0.035,Y -175.888,Z 1552.770,A 0.000,B 0.000,C 90.000,E1 138.528} C_DIS
LIN {X -0.088,Y -181.491,Z 1552.751,A 0.000,B 0.000,C 90.000,E1 135.162} C_DIS
LIN {X 0.048,Y -187.008,Z 1552.732,A 0.000,B 0.000,C 90.000,E1 131.757} C_DIS
LIN {X 0.049,Y -190.125,Z 1552.723,A 0.000,B 0.000,C 90.000,E1 130.092} C_DIS
LIN {X 0.069,Y -195.896,Z 1552.704,A 0.000,B 0.000,C 90.000,E1 126.790} C_DIS
LIN {X 0.026,Y -200.728,Z 1552.691,A 0.000,B 0.000,C 90.000,E1 124.358} C_DIS
LIN {X 0.066,Y -203.379,Z 1552.682,A 0.000,B 0.000,C 90.000,E1 122.832} C_DIS
LIN {X 0.069,Y -319.256,Z 1552.682,A 0.000,B 0.000,C 90.000,E1 122.832} C_DIS
LIN {X -0.015,Y -322.983,Z 1552.682,A 0.000,B 0.000,C 90.000,E1 122.752} C_DIS
LIN {X 0.155,Y -326.073,Z 1552.681,A 0.000,B 0.000,C 90.000,E1 122.546} C_DIS
LIN {X 0.076,Y -329.746,Z 1552.679,A 0.000,B 0.000,C 90.000,E1 122.212} C_DIS
LIN {X 0.121,Y -333.263,Z 1552.676,A 0.000,B 0.000,C 90.000,E1 121.671} C_DIS
LIN {X 0.069,Y -335.928,Z 1552.673,A 0.000,B 0.000,C 90.000,E1 121.052} C_DIS
LIN {X 0.006,Y -347.425,Z 1552.657,A 0.000,B 0.000,C 90.000,E1 118.281} C_DIS
LIN {X 0.096,Y -360.342,Z 1552.642,A 0.000,B 0.000,C 90.000,E1 115.540} C_DIS
LIN {X -0.070,Y -374.784,Z 1552.627,A 0.000,B 0.000,C 90.000,E1 112.898} C_DIS
LIN {X 0.079,Y -389.008,Z 1552.614,A 0.000,B 0.000,C 90.000,E1 110.556} C_DIS
LIN {X -0.053,Y -404.637,Z 1552.602,A 0.000,B 0.000,C 90.000,E1 108.308} C_DIS
LIN {X 0.067,Y -421.778,Z 1552.589,A 0.000,B 0.000,C 90.000,E1 106.079} C_DIS
LIN {X -0.047,Y -440.553,Z 1552.577,A 0.000,B 0.000,C 90.000,E1 103.939} C_DIS
LIN {X 0.099,Y -460.487,Z 1552.566,A 0.000,B 0.000,C 90.000,E1 101.883} C_DIS
LIN {X 0.049,Y -483.586,Z 1552.554,A 0.000,B 0.000,C 90.000,E1 99.792} C_DIS
LIN {X -0.072,Y -491.406,Z 1552.551,A 0.000,B 0.000,C 90.000,E1 99.151} C_DIS
LIN {X 0.101,Y -493.788,Z 1552.550,A 0.000,B 0.000,C 90.000,E1 98.916} C_DIS
LIN {X 0.086,Y -495.682,Z 1552.548,A 0.000,B 0.000,C 90.000,E1 98.690} C_DIS
LIN {X 0.146,Y -497.121,Z 1552.547,A 0.000,B 0.000,C 90.000,E1 98.454} C_DIS
LIN {X -0.089,Y -499.118,Z 1552.544,A 0.000,B 0.000,C 90.000,E1 97.992} C_DIS
LIN {X 0.180,Y -499.956,Z 1552.542,A 0.000,B 0.000,C 90.000,E1 97.473} C_DIS
LIN {X 0.026,Y -499.788,Z 1552.539,A 0.000,B 0.000,C 90.000,E1 97.004} C_DIS
LIN {X -0.187,Y -498.589,Z 1552.536,A 0.000,B 0.000,C 90.000,E1 96.543} C_DIS
LIN {X 0.173,Y -497.546,Z 1552.535,A 0.000,B 0.000,C 90.000,E1 96.258} C_DIS
LIN {X 0.041,Y -496.135,Z 1552.534,A 0.000,B 0.000,C 90.000,E1 96.030} C_DIS
LIN {X -0.004,Y -478.516,Z 1552.518,A 0.000,B 0.000,C 90.000,E1 93.326} C_DIS
LIN {X 0.078,Y -470.414,Z 1552.511,A 0.000,B 0.000,C 90.000,E1 92.064} C_DIS
LIN {X 0.035,Y -461.908,Z 1552.505,A 0.000,B 0.000,C 90.000,E1 90.802} C_DIS
LIN {X -0.132,Y -453.057,Z 1552.497,A 0.000,B 0.000,C 90.000,E1 89.542} C_DIS
LIN {X 0.226,Y -441.916,Z 1552.489,A 0.000,B 0.000,C 90.000,E1 87.936} C_DIS
LIN {X -0.055,Y -430.337,Z 1552.480,A 0.000,B 0.000,C 90.000,E1 86.388} C_DIS
LIN {X 0.060,Y -416.732,Z 1552.469,A 0.000,B 0.000,C 90.000,E1 84.489} C_DIS
LIN {X 0.088,Y -399.726,Z 1552.456,A 0.000,B 0.000,C 90.000,E1 82.008} C_DIS
LIN {X 0.205,Y -381.879,Z 1552.440,A 0.000,B 0.000,C 90.000,E1 79.162} C_DIS
LIN {X 0.021,Y -365.136,Z 1552.424,A 0.000,B 0.000,C 90.000,E1 76.284} C_DIS
LIN {X -0.092,Y -352.198,Z 1552.411,A 0.000,B 0.000,C 90.000,E1 73.921} C_DIS
LIN {X 0.096,Y -341.013,Z 1552.399,A 0.000,B 0.000,C 90.000,E1 71.764} C_DIS
LIN {X 0.085,Y -326.994,Z 1552.383,A 0.000,B 0.000,C 90.000,E1 68.975} C_DIS
LIN {X 0.013,Y -310.922,Z 1552.364,A 0.000,B 0.000,C 90.000,E1 65.485} C_DIS
LIN {X 0.017,Y -300.969,Z 1552.351,A 0.000,B 0.000,C 90.000,E1 63.204} C_DIS
LIN {X 0.064,Y -289.744,Z 1552.336,A 0.000,B 0.000,C 90.000,E1 60.539} C_DIS
LIN {X -0.091,Y -279.964,Z 1552.323,A 0.000,B 0.000,C 90.000,E1 58.201} C_DIS
LIN {X 0.086,Y -267.772,Z 1552.306,A 0.000,B 0.000,C 90.000,E1 55.055} C_DIS
LIN {X -0.100,Y -257.312,Z 1552.290,A 0.000,B 0.000,C 90.000,E1 52.271} C_DIS
LIN {X -0.052,Y -246.023,Z 1552.272,A 0.000,B 0.000,C 90.000,E1 49.013} C_DIS
LIN {X 0.142,Y -235.492,Z 1552.254,A 0.000,B 0.000,C 90.000,E1 45.648} C_DIS
LIN {X -0.051,Y -226.960,Z 1552.237,A 0.000,B 0.000,C 90.000,E1 42.690} C_DIS
LIN {X -0.085,Y -219.227,Z 1552.220,A 0.000,B 0.000,C 90.000,E1 39.644} C_DIS
LIN {X 0.051,Y -212.208,Z 1552.203,A 0.000,B 0.000,C 90.000,E1 36.503} C_DIS
LIN {X -0.022,Y -205.998,Z 1552.185,A 0.000,B 0.000,C 90.000,E1 33.372} C_DIS
LIN {X -0.016,Y -200.534,Z 1552.168,A 0.000,B 0.000,C 90.000,E1 30.178} C_DIS
LIN {X 0.089,Y -194.778,Z 1552.145,A 0.000,B 0.000,C 90.000,E1 26.104} C_DIS
LIN {X 0.039,Y -190.049,Z 1552.122,A 0.000,B 0.000,C 90.000,E1 22.025} C_DIS
LIN {X 0.090,Y -186.021,Z 1552.099,A 0.000,B 0.000,C 90.000,E1 17.873} C_DIS
LIN {X 0.023,Y -182.127,Z 1552.072,A 0.000,B 0.000,C 90.000,E1 12.883} C_DIS
LIN {X 0.074,Y -179.169,Z 1552.044,A 0.000,B 0.000,C 90.000,E1 7.814} C_DIS
LIN {X 0.000,Y -176.873,Z 1552.000,A 0.000,B 0.000,C 90.000,E1 360.000} C_DIS
LIN {X -0.057,Y -178.313,Z 1551.941,A 0.000,B 0.000,C 90.000,E1 349.342} C_DIS
LIN {X 0.094,Y -180.904,Z 1551.912,A 0.000,B 0.000,C 90.000,E1 344.212} C_DIS
LIN {X -0.089,Y -184.218,Z 1551.889,A 0.000,B 0.000,C 90.000,E1 340.061} C_DIS
LIN {X -0.036,Y -188.436,Z 1551.866,A 0.000,B 0.000,C 90.000,E1 335.869} C_DIS
LIN {X 0.019,Y -193.624,Z 1551.843,A 0.000,B 0.000,C 90.000,E1 331.719} C_DIS
LIN {X -0.073,Y -199.716,Z 1551.820,A 0.000,B 0.000,C 90.000,E1 327.661} C_DIS
LIN {X 0.038,Y -205.423,Z 1551.802,A 0.000,B 0.000,C 90.000,E1 324.402} C_DIS
LIN {X -0.089,Y -211.846,Z 1551.785,A 0.000,B 0.000,C 90.000,E1 321.251} C_DIS
LIN {X 0.015,Y -219.183,Z 1551.767,A 0.000,B 0.000,C 90.000,E1 318.081} C_DIS
LIN {X 0.075,Y -228.315,Z 1551.748,A 0.000,B 0.000,C 90.000,E1 314.595} C_DIS
LIN {X -0.033,Y -237.499,Z 1551.731,A 0.000,B 0.000,C 90.000,E1 311.595} C_DIS
LIN {X -0.001,Y -244.000,Z 1551.721,A 0.000,B 0.000,C 90.000,E1 309.725} C_DIS
LIN {X -0.020,Y -249.918,Z 1551.713,A 0.000,B 0.000,C 90.000,E1 308.257} C_DIS
LIN {X 0.035,Y -256.525,Z 1551.704,A 0.000,B 0.000,C 90.000,E1 306.790} C_DIS
LIN {X -0.087,Y -265.762,Z 1551.694,A 0.000,B 0.000,C 90.000,E1 305.025} C_DIS
LIN {X 0.081,Y -273.996,Z 1551.687,A 0.000,B 0.000,C 90.000,E1 303.579} C_DIS
LIN {X -0.112,Y -287.528,Z 1551.675,A 0.000,B 0.000,C 90.000,E1 301.544} C_DIS
LIN {X 0.110,Y -309.643,Z 1551.658,A 0.000,B 0.000,C 90.000,E1 298.487} C_DIS
LIN {X -0.001,Y -324.943,Z 1551.648,A 0.000,B 0.000,C 90.000,E1 296.565} C_DIS
LIN {X -0.087,Y -342.962,Z 1551.635,A 0.000,B 0.000,C 90.000,E1 294.387} C_DIS
LIN {X 0.082,Y -363.925,Z 1551.622,A 0.000,B 0.000,C 90.000,E1 291.972} C_DIS
LIN {X 0.123,Y -376.854,Z 1551.614,A 0.000,B 0.000,C 90.000,E1 290.556} C_DIS
LIN {X -0.129,Y -387.004,Z 1551.608,A 0.000,B 0.000,C 90.000,E1 289.450} C_DIS
LIN {X 0.192,Y -394.196,Z 1551.603,A 0.000,B 0.000,C 90.000,E1 288.544} C_DIS
LIN {X 0.201,Y -400.780,Z 1551.599,A 0.000,B 0.000,C 90.000,E1 287.692} C_DIS
LIN {X 0.157,Y -406.642,Z 1551.594,A 0.000,B 0.000,C 90.000,E1 286.858} C_DIS
LIN {X 0.062,Y -410.138,Z 1551.591,A 0.000,B 0.000,C 90.000,E1 286.315} C_DIS
LIN {X 0.096,Y -414.718,Z 1551.586,A 0.000,B 0.000,C 90.000,E1 285.481} C_DIS
LIN {X 0.070,Y -418.405,Z 1551.582,A 0.000,B 0.000,C 90.000,E1 284.662} C_DIS
LIN {X 0.183,Y -421.351,Z 1551.577,A 0.000,B 0.000,C 90.000,E1 283.828} C_DIS
LIN {X 0.065,Y -422.896,Z 1551.574,A 0.000,B 0.000,C 90.000,E1 283.300} C_DIS
LIN {X -0.042,Y -423.988,Z 1551.571,A 0.000,B 0.000,C 90.000,E1 282.771} C_DIS
LIN {X -0.140,Y -424.661,Z 1551.568,A 0.000,B 0.000,C 90.000,E1 282.243} C_DIS
LIN {X -0.232,Y -424.839,Z 1551.565,A 0.000,B 0.000,C 90.000,E1 281.715} C_DIS
LIN {X 0.096,Y -424.511,Z 1551.562,A 0.000,B 0.000,C 90.000,E1 281.130} C_DIS
LIN {X 0.007,Y -423.655,Z 1551.559,A 0.000,B 0.000,C 90.000,E1 280.602} C_DIS
LIN {X -0.085,Y -422.192,Z 1551.556,A 0.000,B 0.000,C 90.000,E1 280.074} C_DIS
LIN {X 0.160,Y -420.142,Z 1551.553,A 0.000,B 0.000,C 90.000,E1 279.500} C_DIS
LIN {X 0.051,Y -417.286,Z 1551.550,A 0.000,B 0.000,C 90.000,E1 278.973} C_DIS
LIN {X -0.141,Y -413.655,Z 1551.547,A 0.000,B 0.000,C 90.000,E1 278.454} C_DIS
LIN {X 0.117,Y -409.212,Z 1551.544,A 0.000,B 0.000,C 90.000,E1 277.871} C_DIS
LIN {X -0.112,Y -403.867,Z 1551.541,A 0.000,B 0.000,C 90.000,E1 277.352} C_DIS
LIN {X -0.102,Y -397.973,Z 1551.538,A 0.000,B 0.000,C 90.000,E1 276.834} C_DIS
LIN {X -0.087,Y -392.090,Z 1551.535,A 0.000,B 0.000,C 90.000,E1 276.372} C_DIS
LIN {X 0.180,Y -385.833,Z 1551.533,A 0.000,B 0.000,C 90.000,E1 275.910} C_DIS
LIN {X -0.049,Y -379.705,Z 1551.531,A 0.000,B 0.000,C 90.000,E1 275.568} C_DIS
LIN {X -0.064,Y -373.200,Z 1551.529,A 0.000,B 0.000,C 90.000,E1 275.220} C_DIS
LIN {X -0.087,Y -363.493,Z 1551.526,A 0.000,B 0.000,C 90.000,E1 274.759} C_DIS
LIN {X 0.029,Y -350.748,Z 1551.523,A 0.000,B 0.000,C 90.000,E1 274.188} C_DIS
LIN {X 0.028,Y -337.874,Z 1551.520,A 0.000,B 0.000,C 90.000,E1 273.669} C_DIS
LIN {X 0.032,Y -324.719,Z 1551.518,A 0.000,B 0.000,C 90.000,E1 273.212} C_DIS
LIN {X -0.071,Y -314.321,Z 1551.516,A 0.000,B 0.000,C 90.000,E1 272.922} C_DIS
LIN {X 0.086,Y -304.254,Z 1551.515,A 0.000,B 0.000,C 90.000,E1 272.636} C_DIS
LIN {X 0.081,Y -292.953,Z 1551.513,A 0.000,B 0.000,C 90.000,E1 272.407} C_DIS
LIN {X 0.031,Y -279.923,Z 1551.512,A 0.000,B 0.000,C 90.000,E1 272.236} C_DIS
LIN {X -0.029,Y -266.234,Z 1551.512,A 0.000,B 0.000,C 90.000,E1 272.121} C_DIS
LIN {X -0.023,Y -253.965,Z 1551.511,A 0.000,B 0.000,C 90.000,E1 272.064} C_DIS
LIN {X -0.049,Y -181.254,Z 1551.511,A 0.000,B 0.000,C 90.000,E1 272.064} C_DIS
LIN {X -0.070,Y -181.580,Z 1551.502,A 0.000,B 0.000,C 90.000,E1 270.344} C_DIS
LIN {X -0.094,Y -180.901,Z 1551.474,A 0.000,B 0.000,C 90.000,E1 265.298} C_DIS
LIN {X 0.035,Y -180.230,Z 1551.464,A 0.000,B 0.000,C 90.000,E1 263.571} C_DIS
LIN {X -0.012,Y -179.042,Z 1551.446,A 0.000,B 0.000,C 90.000,E1 260.208} C_DIS
LIN {X 0.051,Y -178.713,Z 1551.441,A 0.000,B 0.000,C 90.000,E1 259.342} C_DIS
LIN {X -0.056,Y -175.761,Z 1551.413,A 0.000,B 0.000,C 90.000,E1 254.283} C_DIS
LIN {X -0.006,Y -171.945,Z 1551.384,A 0.000,B 0.000,C 90.000,E1 249.135} C_DIS
LIN {X -0.030,Y -171.330,Z 1551.379,A 0.000,B 0.000,C 90.000,E1 248.284} C_DIS
LIN {X 0.023,Y -167.586,Z 1551.355,A 0.000,B 0.000,C 90.000,E1 243.948} C_DIS
LIN {X -0.039,Y -166.222,Z 1551.346,A 0.000,B 0.000,C 90.000,E1 242.231} C_DIS
LIN {X -0.050,Y -162.984,Z 1551.326,A 0.000,B 0.000,C 90.000,E1 238.742} C_DIS
LIN {X -0.002,Y -160.900,Z 1551.312,A 0.000,B 0.000,C 90.000,E1 236.087} C_DIS
LIN {X -0.025,Y -157.667,Z 1551.292,A 0.000,B 0.000,C 90.000,E1 232.557} C_DIS
LIN {X -0.086,Y -155.705,Z 1551.277,A 0.000,B 0.000,C 90.000,E1 229.908} C_DIS
LIN {X -0.031,Y -151.968,Z 1551.252,A 0.000,B 0.000,C 90.000,E1 225.405} C_DIS
LIN {X -0.015,Y -150.210,Z 1551.237,A 0.000,B 0.000,C 90.000,E1 222.690} C_DIS
LIN {X -0.090,Y -146.976,Z 1551.212,A 0.000,B 0.000,C 90.000,E1 218.177} C_DIS
LIN {X 0.019,Y -145.562,Z 1551.197,A 0.000,B 0.000,C 90.000,E1 215.391} C_DIS
LIN {X 0.018,Y -142.954,Z 1551.171,A 0.000,B 0.000,C 90.000,E1 210.797} C_DIS
LIN {X -0.051,Y -141.580,Z 1551.151,A 0.000,B 0.000,C 90.000,E1 207.129} C_DIS
LIN {X -0.003,Y -139.415,Z 1551.115,A 0.000,B 0.000,C 90.000,E1 200.610} C_DIS
LIN {X 0.048,Y -139.140,Z 1551.104,A 0.000,B 0.000,C 90.000,E1 198.725} C_DIS
LIN {X -0.061,Y -138.348,Z 1551.057,A 0.000,B 0.000,C 90.000,E1 190.366} C_DIS
LIN {X 0.063,Y -139.492,Z 1551.006,A 0.000,B 0.000,C 90.000,E1 180.974} C_DIS
LIN {X 0.005,Y -141.103,Z 1550.974,A 0.000,B 0.000,C 90.000,E1 175.412} C_DIS
LIN {X -0.042,Y -142.482,Z 1550.959,A 0.000,B 0.000,C 90.000,E1 172.648} C_DIS
LIN {X 0.047,Y -144.731,Z 1550.933,A 0.000,B 0.000,C 90.000,E1 167.993} C_DIS
LIN {X -0.003,Y -147.335,Z 1550.913,A 0.000,B 0.000,C 90.000,E1 164.338} C_DIS
LIN {X 0.062,Y -150.658,Z 1550.888,A 0.000,B 0.000,C 90.000,E1 159.752} C_DIS
LIN {X -0.056,Y -154.136,Z 1550.868,A 0.000,B 0.000,C 90.000,E1 156.177} C_DIS
LIN {X 0.006,Y -157.565,Z 1550.848,A 0.000,B 0.000,C 90.000,E1 152.564} C_DIS
LIN {X 0.030,Y -161.808,Z 1550.828,A 0.000,B 0.000,C 90.000,E1 148.997} C_DIS
LIN {X 0.050,Y -166.000,Z 1550.808,A 0.000,B 0.000,C 90.000,E1 145.468} C_DIS
LIN {X 0.043,Y -170.998,Z 1550.789,A 0.000,B 0.000,C 90.000,E1 141.984} C_DIS
LIN {X -0.042,Y -175.868,Z 1550.770,A 0.000,B 0.000,C 90.000,E1 138.566} C_DIS
LIN {X -0.049,Y -181.473,Z 1550.751,A 0.000,B 0.000,C 90.000,E1 135.162} C_DIS
LIN {X 0.089,Y -186.985,Z 1550.732,A 0.000,B 0.000,C 90.000,E1 131.757} C_DIS
LIN {X 0.091,Y -190.101,Z 1550.723,A 0.000,B 0.000,C 90.000,E1 130.092} C_DIS
LIN {X 0.110,Y -195.874,Z 1550.705,A 0.000,B 0.000,C 90.000,E1 126.790} C_DIS
LIN {X -0.098,Y -200.705,Z 1550.691,A 0.000,B 0.000,C 90.000,E1 124.405} C_DIS
LIN {X 0.032,Y -203.309,Z 1550.683,A 0.000,B 0.000,C 90.000,E1 122.880} C_DIS
LIN {X 0.015,Y -318.882,Z 1550.683,A 0.000,B 0.000,C 90.000,E1 122.880} C_DIS
LIN {X 0.052,Y -323.378,Z 1550.682,A 0.000,B 0.000,C 90.000,E1 122.752} C_DIS
LIN {X 0.156,Y -326.395,Z 1550.681,A 0.000,B 0.000,C 90.000,E1 122.546} C_DIS
LIN {X -0.087,Y -330.110,Z 1550.679,A 0.000,B 0.000,C 90.000,E1 122.212} C_DIS
LIN {X -0.205,Y -333.567,Z 1550.676,A 0.000,B 0.000,C 90.000,E1 121.671} C_DIS
LIN {X 0.010,Y -338.564,Z 1550.669,A 0.000,B 0.000,C 90.000,E1 120.384} C_DIS
LIN {X -0.147,Y -350.394,Z 1550.653,A 0.000,B 0.000,C 90.000,E1 117.641} C_DIS
LIN {X 0.026,Y -363.671,Z 1550.638,A 0.000,B 0.000,C 90.000,E1 114.899} C_DIS
LIN {X -0.056,Y -378.501,Z 1550.624,A 0.000,B 0.000,C 90.000,E1 112.259} C_DIS
LIN {X 0.039,Y -393.098,Z 1550.611,A 0.000,B 0.000,C 90.000,E1 109.939} C_DIS
LIN {X 0.000,Y -409.127,Z 1550.598,A 0.000,B 0.000,C 90.000,E1 107.692} C_DIS
LIN {X 0.104,Y -426.701,Z 1550.586,A 0.000,B 0.000,C 90.000,E1 105.481} C_DIS
LIN {X 0.040,Y -445.896,Z 1550.574,A 0.000,B 0.000,C 90.000,E1 103.355} C_DIS
LIN {X 0.023,Y -465.990,Z 1550.563,A 0.000,B 0.000,C 90.000,E1 101.366} C_DIS
LIN {X -0.017,Y -489.242,Z 1550.552,A 0.000,B 0.000,C 90.000,E1 99.321} C_DIS
LIN {X 0.080,Y -491.849,Z 1550.551,A 0.000,B 0.000,C 90.000,E1 99.095} C_DIS
LIN {X -0.231,Y -494.095,Z 1550.549,A 0.000,B 0.000,C 90.000,E1 98.916} C_DIS
LIN {X 0.248,Y -495.940,Z 1550.548,A 0.000,B 0.000,C 90.000,E1 98.624} C_DIS
LIN {X 0.165,Y -497.333,Z 1550.547,A 0.000,B 0.000,C 90.000,E1 98.398} C_DIS
LIN {X -0.068,Y -499.169,Z 1550.544,A 0.000,B 0.000,C 90.000,E1 97.936} C_DIS
LIN {X 0.267,Y -499.878,Z 1550.541,A 0.000,B 0.000,C 90.000,E1 97.409} C_DIS
LIN {X 0.049,Y -499.586,Z 1550.539,A 0.000,B 0.000,C 90.000,E1 96.947} C_DIS
LIN {X -0.165,Y -498.249,Z 1550.536,A 0.000,B 0.000,C 90.000,E1 96.486} C_DIS
LIN {X 0.196,Y -497.122,Z 1550.535,A 0.000,B 0.000,C 90.000,E1 96.201} C_DIS
LIN {X -0.161,Y -492.232,Z 1550.531,A 0.000,B 0.000,C 90.000,E1 95.511} C_DIS
LIN {X 0.004,Y -478.041,Z 1550.518,A 0.000,B 0.000,C 90.000,E1 93.269} C_DIS
LIN {X 0.080,Y -469.921,Z 1550.511,A 0.000,B 0.000,C 90.000,E1 92.007} C_DIS
LIN {X 0.030,Y -461.403,Z 1550.504,A 0.000,B 0.000,C 90.000,E1 90.745} C_DIS
LIN {X -0.143,Y -452.548,Z 1550.497,A 0.000,B 0.000,C 90.000,E1 89.484} C_DIS
LIN {X 0.013,Y -443.287,Z 1550.490,A 0.000,B 0.000,C 90.000,E1 88.165} C_DIS
LIN {X 0.195,Y -431.785,Z 1550.481,A 0.000,B 0.000,C 90.000,E1 86.560} C_DIS
LIN {X -0.116,Y -418.200,Z 1550.471,A 0.000,B 0.000,C 90.000,E1 84.723} C_DIS
LIN {X -0.056,Y -401.137,Z 1550.457,A 0.000,B 0.000,C 90.000,E1 82.243} C_DIS
LIN {X 0.101,Y -383.219,Z 1550.441,A 0.000,B 0.000,C 90.000,E1 79.398} C_DIS
LIN {X -0.056,Y -364.767,Z 1550.423,A 0.000,B 0.000,C 90.000,E1 76.228} C_DIS
LIN {X -0.081,Y -351.848,Z 1550.410,A 0.000,B 0.000,C 90.000,E1 73.850} C_DIS
LIN {X 0.099,Y -342.253,Z 1550.400,A 0.000,B 0.000,C 90.000,E1 72.000} C_DIS
LIN {X 0.096,Y -326.649,Z 1550.383,A 0.000,B 0.000,C 90.000,E1 68.901} C_DIS
LIN {X 0.021,Y -310.566,Z 1550.363,A 0.000,B 0.000,C 90.000,E1 65.409} C_DIS
LIN {X -0.003,Y -302.050,Z 1550.353,A 0.000,B 0.000,C 90.000,E1 63.461} C_DIS
LIN {X 0.077,Y -292.210,Z 1550.340,A 0.000,B 0.000,C 90.000,E1 61.129} C_DIS
LIN {X -0.025,Y -282.448,Z 1550.327,A 0.000,B 0.000,C 90.000,E1 58.791} C_DIS
LIN {X 0.076,Y -270.147,Z 1550.309,A 0.000,B 0.000,C 90.000,E1 55.674} C_DIS
LIN {X 0.103,Y -260.933,Z 1550.296,A 0.000,B 0.000,C 90.000,E1 53.210} C_DIS
LIN {X 0.089,Y -249.495,Z 1550.278,A 0.000,B 0.000,C 90.000,E1 49.989} C_DIS
LIN {X 0.047,Y -238.754,Z 1550.260,A 0.000,B 0.000,C 90.000,E1 46.701} C_DIS
LIN {X 0.038,Y -228.926,Z 1550.241,A 0.000,B 0.000,C 90.000,E1 43.338} C_DIS
LIN {X 0.030,Y -221.039,Z 1550.224,A 0.000,B 0.000,C 90.000,E1 40.297} C_DIS
LIN {X -0.093,Y -213.867,Z 1550.207,A 0.000,B 0.000,C 90.000,E1 37.237} C_DIS
LIN {X 0.002,Y -207.517,Z 1550.189,A 0.000,B 0.000,C 90.000,E1 34.072} C_DIS
LIN {X 0.051,Y -201.893,Z 1550.172,A 0.000,B 0.000,C 90.000,E1 30.875} C_DIS
LIN {X -0.049,Y -195.998,Z 1550.149,A 0.000,B 0.000,C 90.000,E1 26.873} C_DIS
LIN {X 0.020,Y -191.106,Z 1550.127,A 0.000,B 0.000,C 90.000,E1 22.770} C_DIS
LIN {X -0.068,Y -186.947,Z 1550.104,A 0.000,B 0.000,C 90.000,E1 18.671} C_DIS
LIN {X 0.006,Y -182.900,Z 1550.076,A 0.000,B 0.000,C 90.000,E1 13.647} C_DIS
LIN {X -0.060,Y -179.818,Z 1550.048,A 0.000,B 0.000,C 90.000,E1 8.624} C_DIS
LIN {X -0.013,Y -177.411,Z 1550.010,A 0.000,B 0.000,C 90.000,E1 1.835} C_DIS
LIN {X -0.038,Y -178.583,Z 1549.941,A 0.000,B 0.000,C 90.000,E1 349.342} C_DIS
LIN {X -0.051,Y -181.179,Z 1549.912,A 0.000,B 0.000,C 90.000,E1 344.267} C_DIS
LIN {X -0.051,Y -184.462,Z 1549.889,A 0.000,B 0.000,C 90.000,E1 340.061} C_DIS
LIN {X 0.010,Y -188.658,Z 1549.866,A 0.000,B 0.000,C 90.000,E1 335.869} C_DIS
LIN {X -0.097,Y -193.851,Z 1549.843,A 0.000,B 0.000,C 90.000,E1 331.769} C_DIS
LIN {X -0.009,Y -199.908,Z 1549.820,A 0.000,B 0.000,C 90.000,E1 327.661} C_DIS
LIN {X 0.107,Y -205.550,Z 1549.802,A 0.000,B 0.000,C 90.000,E1 324.402} C_DIS
LIN {X -0.014,Y -211.965,Z 1549.785,A 0.000,B 0.000,C 90.000,E1 321.251} C_DIS
LIN {X 0.096,Y -219.263,Z 1549.767,A 0.000,B 0.000,C 90.000,E1 318.081} C_DIS
LIN {X -0.001,Y -228.352,Z 1549.748,A 0.000,B 0.000,C 90.000,E1 314.636} C_DIS
LIN {X 0.057,Y -237.502,Z 1549.731,A 0.000,B 0.000,C 90.000,E1 311.595} C_DIS
LIN {X 0.091,Y -243.983,Z 1549.721,A 0.000,B 0.000,C 90.000,E1 309.725} C_DIS
LIN {X 0.075,Y -249.845,Z 1549.713,A 0.000,B 0.000,C 90.000,E1 308.257} C_DIS
LIN {X 0.132,Y -256.428,Z 1549.705,A 0.000,B 0.000,C 90.000,E1 306.790} C_DIS
LIN {X 0.011,Y -265.643,Z 1549.695,A 0.000,B 0.000,C 90.000,E1 305.025} C_DIS
LIN {X -0.048,Y -273.838,Z 1549.687,A 0.000,B 0.000,C 90.000,E1 303.627} C_DIS
LIN {X 0.026,Y -284.992,Z 1549.677,A 0.000,B 0.000,C 90.000,E1 301.878} C_DIS
LIN {X -0.080,Y -306.897,Z 1549.660,A 0.000,B 0.000,C 90.000,E1 298.871} C_DIS
LIN {X 0.178,Y -322.197,Z 1549.649,A 0.000,B 0.000,C 90.000,E1 296.873} C_DIS
LIN {X -0.032,Y -337.518,Z 1549.639,A 0.000,B 0.000,C 90.000,E1 295.027} C_DIS
LIN {X -0.066,Y -353.190,Z 1549.629,A 0.000,B 0.000,C 90.000,E1 293.206} C_DIS
LIN {X -0.066,Y -369.040,Z 1549.619,A 0.000,B 0.000,C 90.000,E1 291.461} C_DIS
LIN {X 0.098,Y -379.416,Z 1549.613,A 0.000,B 0.000,C 90.000,E1 290.301} C_DIS
LIN {X 0.085,Y -387.000,Z 1549.608,A 0.000,B 0.000,C 90.000,E1 289.450} C_DIS
LIN {X 0.034,Y -394.191,Z 1549.603,A 0.000,B 0.000,C 90.000,E1 288.598} C_DIS
LIN {X -0.082,Y -400.809,Z 1549.599,A 0.000,B 0.000,C 90.000,E1 287.764} C_DIS
LIN {X -0.010,Y -406.715,Z 1549.594,A 0.000,B 0.000,C 90.000,E1 286.913} C_DIS
LIN {X -0.009,Y -411.879,Z 1549.589,A 0.000,B 0.000,C 90.000,E1 286.079} C_DIS
LIN {X -0.075,Y -414.852,Z 1549.586,A 0.000,B 0.000,C 90.000,E1 285.536} C_DIS
LIN {X -0.103,Y -418.600,Z 1549.582,A 0.000,B 0.000,C 90.000,E1 284.717} C_DIS
LIN {X 0.010,Y -421.571,Z 1549.577,A 0.000,B 0.000,C 90.000,E1 283.883} C_DIS
LIN {X -0.109,Y -423.145,Z 1549.574,A 0.000,B 0.000,C 90.000,E1 283.355} C_DIS
LIN {X -0.217,Y -424.330,Z 1549.571,A 0.000,B 0.000,C 90.000,E1 282.827} C_DIS
LIN {X 0.101,Y -425.082,Z 1549.568,A 0.000,B 0.000,C 90.000,E1 282.243} C_DIS
LIN {X 0.011,Y -425.331,Z 1549.565,A 0.000,B 0.000,C 90.000,E1 281.715} C_DIS
LIN {X -0.075,Y -425.075,Z 1549.562,A 0.000,B 0.000,C 90.000,E1 281.186} C_DIS
LIN {X -0.162,Y -424.233,Z 1549.559,A 0.000,B 0.000,C 90.000,E1 280.658} C_DIS
LIN {X 0.165,Y -422.906,Z 1549.556,A 0.000,B 0.000,C 90.000,E1 280.074} C_DIS
LIN {X -0.002,Y -420.890,Z 1549.553,A 0.000,B 0.000,C 90.000,E1 279.557} C_DIS
LIN {X -0.107,Y -418.122,Z 1549.550,A 0.000,B 0.000,C 90.000,E1 279.029} C_DIS
LIN {X 0.117,Y -414.600,Z 1549.547,A 0.000,B 0.000,C 90.000,E1 278.454} C_DIS
LIN {X -0.085,Y -410.189,Z 1549.544,A 0.000,B 0.000,C 90.000,E1 277.936} C_DIS
LIN {X 0.150,Y -404.908,Z 1549.541,A 0.000,B 0.000,C 90.000,E1 277.352} C_DIS
LIN {X 0.118,Y -399.063,Z 1549.538,A 0.000,B 0.000,C 90.000,E1 276.834} C_DIS
LIN {X 0.056,Y -393.032,Z 1549.535,A 0.000,B 0.000,C 90.000,E1 276.372} C_DIS
LIN {X -0.058,Y -386.866,Z 1549.533,A 0.000,B 0.000,C 90.000,E1 275.967} C_DIS
LIN {X 0.020,Y -380.487,Z 1549.531,A 0.000,B 0.000,C 90.000,E1 275.568} C_DIS
LIN {X 0.010,Y -373.988,Z 1549.529,A 0.000,B 0.000,C 90.000,E1 275.220} C_DIS
LIN {X -0.004,Y -364.304,Z 1549.526,A 0.000,B 0.000,C 90.000,E1 274.759} C_DIS
LIN {X 0.104,Y -351.527,Z 1549.523,A 0.000,B 0.000,C 90.000,E1 274.188} C_DIS
LIN {X 0.108,Y -338.739,Z 1549.521,A 0.000,B 0.000,C 90.000,E1 273.669} C_DIS
LIN {X 0.088,Y -325.425,Z 1549.518,A 0.000,B 0.000,C 90.000,E1 273.212} C_DIS
LIN {X 0.005,Y -315.203,Z 1549.516,A 0.000,B 0.000,C 90.000,E1 272.922} C_DIS
LIN {X 0.137,Y -305.019,Z 1549.515,A 0.000,B 0.000,C 90.000,E1 272.636} C_DIS
LIN {X 0.129,Y -293.919,Z 1549.514,A 0.000,B 0.000,C 90.000,E1 272.407} C_DIS
LIN {X 0.065,Y -280.969,Z 1549.512,A 0.000,B 0.000,C 90.000,E1 272.236} C_DIS
LIN {X 0.001,Y -267.191,Z 1549.512,A 0.000,B 0.000,C 90.000,E1 272.121} C_DIS
LIN {X 0.008,Y -255.392,Z 1549.511,A 0.000,B 0.000,C 90.000,E1 272.064} C_DIS
LIN {X -0.027,Y -181.253,Z 1549.511,A 0.000,B 0.000,C 90.000,E1 272.064} C_DIS
LIN {X -0.047,Y -181.580,Z 1549.502,A 0.000,B 0.000,C 90.000,E1 270.344} C_DIS
LIN {X -0.072,Y -180.903,Z 1549.474,A 0.000,B 0.000,C 90.000,E1 265.298} C_DIS
LIN {X 0.058,Y -180.233,Z 1549.464,A 0.000,B 0.000,C 90.000,E1 263.571} C_DIS
LIN {X 0.073,Y -178.717,Z 1549.441,A 0.000,B 0.000,C 90.000,E1 259.342} C_DIS
LIN {X -0.034,Y -175.765,Z 1549.413,A 0.000,B 0.000,C 90.000,E1 254.283} C_DIS
LIN {X 0.016,Y -171.949,Z 1549.384,A 0.000,B 0.000,C 90.000,E1 249.135} C_DIS
LIN {X -0.008,Y -171.337,Z 1549.379,A 0.000,B 0.000,C 90.000,E1 248.284} C_DIS
LIN {X -0.029,Y -167.591,Z 1549.355,A 0.000,B 0.000,C 90.000,E1 243.973} C_DIS
LIN {X -0.017,Y -166.229,Z 1549.346,A 0.000,B 0.000,C 90.000,E1 242.231} C_DIS
LIN {X -0.029,Y -162.989,Z 1549.326,A 0.000,B 0.000,C 90.000,E1 238.742} C_DIS
LIN {X 0.019,Y -160.907,Z 1549.312,A 0.000,B 0.000,C 90.000,E1 236.087} C_DIS
LIN {X -0.004,Y -157.672,Z 1549.292,A 0.000,B 0.000,C 90.000,E1 232.557} C_DIS
LIN {X -0.066,Y -155.711,Z 1549.277,A 0.000,B 0.000,C 90.000,E1 229.908} C_DIS
LIN {X -0.011,Y -151.973,Z 1549.252,A 0.000,B 0.000,C 90.000,E1 225.405} C_DIS
LIN {X 0.005,Y -150.216,Z 1549.237,A 0.000,B 0.000,C 90.000,E1 222.690} C_DIS
LIN {X -0.070,Y -146.980,Z 1549.212,A 0.000,B 0.000,C 90.000,E1 218.177} C_DIS
LIN {X 0.039,Y -145.566,Z 1549.197,A 0.000,B 0.000,C 90.000,E1 215.391} C_DIS
LIN {X 0.038,Y -142.958,Z 1549.171,A 0.000,B 0.000,C 90.000,E1 210.797} C_DIS
LIN {X -0.032,Y -141.584,Z 1549.151,A 0.000,B 0.000,C 90.000,E1 207.129} C_DIS
LIN {X 0.015,Y -139.417,Z 1549.115,A 0.000,B 0.000,C 90.000,E1 200.610} C_DIS
LIN {X 0.068,Y -139.142,Z 1549.104,A 0.000,B 0.000,C 90.000,E1 198.725} C_DIS
LIN {X -0.042,Y -138.348,Z 1549.057,A 0.000,B 0.000,C 90.000,E1 190.366} C_DIS
LIN {X -0.056,Y -139.491,Z 1549.006,A 0.000,B 0.000,C 90.000,E1 181.031} C_DIS
LIN {X 0.024,Y -141.099,Z 1548.975,A 0.000,B 0.000,C 90.000,E1 175.412} C_DIS
LIN {X -0.023,Y -142.478,Z 1548.959,A 0.000,B 0.000,C 90.000,E1 172.648} C_DIS
LIN {X 0.066,Y -144.726,Z 1548.933,A 0.000,B 0.000,C 90.000,E1 167.993} C_DIS
LIN {X 0.017,Y -147.330,Z 1548.913,A 0.000,B 0.000,C 90.000,E1 164.338} C_DIS
LIN {X 0.083,Y -150.652,Z 1548.888,A 0.000,B 0.000,C 90.000,E1 159.752} C_DIS
LIN {X -0.035,Y -154.129,Z 1548.868,A 0.000,B 0.000,C 90.000,E1 156.177} C_DIS
LIN {X 0.027,Y -157.556,Z 1548.848,A 0.000,B 0.000,C 90.000,E1 152.564} C_DIS
LIN {X 0.052,Y -161.799,Z 1548.828,A 0.000,B 0.000,C 90.000,E1 148.997} C_DIS
LIN {X 0.071,Y -165.991,Z 1548.808,A 0.000,B 0.000,C 90.000,E1 145.468} C_DIS
LIN {X 0.065,Y -170.987,Z 1548.789,A 0.000,B 0.000,C 90.000,E1 141.984} C_DIS
LIN {X -0.020,Y -175.857,Z 1548.770,A 0.000,B 0.000,C 90.000,E1 138.566} C_DIS
LIN {X -0.026,Y -181.462,Z 1548.751,A 0.000,B 0.000,C 90.000,E1 135.162} C_DIS
LIN {X 0.111,Y -186.973,Z 1548.732,A 0.000,B 0.000,C 90.000,E1 131.757} C_DIS
LIN {X 0.114,Y -190.088,Z 1548.723,A 0.000,B 0.000,C 90.000,E1 130.092} C_DIS
LIN {X 0.016,Y -195.861,Z 1548.705,A 0.000,B 0.000,C 90.000,E1 126.824} C_DIS
LIN {X -0.074,Y -200.692,Z 1548.691,A 0.000,B 0.000,C 90.000,E1 124.405} C_DIS
LIN {X -0.130,Y -203.249,Z 1548.683,A 0.000,B 0.000,C 90.000,E1 122.959} C_DIS
LIN {X 0.028,Y -319.127,Z 1548.683,A 0.000,B 0.000,C 90.000,E1 122.911} C_DIS
LIN {X 0.091,Y -323.816,Z 1548.682,A 0.000,B 0.000,C 90.000,E1 122.752} C_DIS
LIN {X 0.062,Y -326.886,Z 1548.681,A 0.000,B 0.000,C 90.000,E1 122.546} C_DIS
LIN {X 0.075,Y -330.608,Z 1548.679,A 0.000,B 0.000,C 90.000,E1 122.133} C_DIS
LIN {X -0.175,Y -332.497,Z 1548.677,A 0.000,B 0.000,C 90.000,E1 121.878} C_DIS
LIN {X 0.032,Y -333.977,Z 1548.675,A 0.000,B 0.000,C 90.000,E1 121.544} C_DIS
LIN {X 0.087,Y -346.638,Z 1548.658,A 0.000,B 0.000,C 90.000,E1 118.437} C_DIS
LIN {X 0.006,Y -359.462,Z 1548.643,A 0.000,B 0.000,C 90.000,E1 115.720} C_DIS
LIN {X -0.198,Y -373.811,Z 1548.628,A 0.000,B 0.000,C 90.000,E1 113.078} C_DIS
LIN {X -0.083,Y -387.941,Z 1548.615,A 0.000,B 0.000,C 90.000,E1 110.737} C_DIS
LIN {X -0.122,Y -403.470,Z 1548.603,A 0.000,B 0.000,C 90.000,E1 108.471} C_DIS
LIN {X -0.166,Y -420.504,Z 1548.590,A 0.000,B 0.000,C 90.000,E1 106.260} C_DIS
LIN {X 0.108,Y -439.162,Z 1548.578,A 0.000,B 0.000,C 90.000,E1 104.064} C_DIS
LIN {X 0.172,Y -459.057,Z 1548.567,A 0.000,B 0.000,C 90.000,E1 102.007} C_DIS
LIN {X 0.031,Y -479.510,Z 1548.556,A 0.000,B 0.000,C 90.000,E1 100.141} C_DIS
LIN {X 0.142,Y -492.491,Z 1548.550,A 0.000,B 0.000,C 90.000,E1 99.029} C_DIS
LIN {X -0.242,Y -494.541,Z 1548.549,A 0.000,B 0.000,C 90.000,E1 98.859} C_DIS
LIN {X 0.158,Y -496.306,Z 1548.548,A 0.000,B 0.000,C 90.000,E1 98.568} C_DIS
LIN {X -0.005,Y -497.626,Z 1548.546,A 0.000,B 0.000,C 90.000,E1 98.341} C_DIS
LIN {X -0.167,Y -499.253,Z 1548.544,A 0.000,B 0.000,C 90.000,E1 97.871} C_DIS
LIN {X 0.101,Y -499.790,Z 1548.541,A 0.000,B 0.000,C 90.000,E1 97.352} C_DIS
LIN {X -0.115,Y -499.330,Z 1548.538,A 0.000,B 0.000,C 90.000,E1 96.891} C_DIS
LIN {X 0.166,Y -497.801,Z 1548.536,A 0.000,B 0.000,C 90.000,E1 96.372} C_DIS
LIN {X 0.031,Y -496.553,Z 1548.534,A 0.000,B 0.000,C 90.000,E1 96.144} C_DIS
LIN {X 0.002,Y -479.006,Z 1548.519,A 0.000,B 0.000,C 90.000,E1 93.440} C_DIS
LIN {X 0.086,Y -470.957,Z 1548.512,A 0.000,B 0.000,C 90.000,E1 92.178} C_DIS
LIN {X -0.155,Y -460.733,Z 1548.504,A 0.000,B 0.000,C 90.000,E1 90.688} C_DIS
LIN {X -0.119,Y -450.074,Z 1548.495,A 0.000,B 0.000,C 90.000,E1 89.141} C_DIS
LIN {X 0.006,Y -440.721,Z 1548.488,A 0.000,B 0.000,C 90.000,E1 87.822} C_DIS
LIN {X 0.139,Y -429.199,Z 1548.479,A 0.000,B 0.000,C 90.000,E1 86.216} C_DIS
LIN {X -0.192,Y -415.615,Z 1548.469,A 0.000,B 0.000,C 90.000,E1 84.375} C_DIS
LIN {X 0.119,Y -400.554,Z 1548.456,A 0.000,B 0.000,C 90.000,E1 82.129} C_DIS
LIN {X -0.093,Y -380.950,Z 1548.439,A 0.000,B 0.000,C 90.000,E1 79.050} C_DIS
LIN {X 0.057,Y -364.256,Z 1548.423,A 0.000,B 0.000,C 90.000,E1 76.117} C_DIS
LIN {X 0.007,Y -351.343,Z 1548.410,A 0.000,B 0.000,C 90.000,E1 73.740} C_DIS
LIN {X -0.155,Y -341.743,Z 1548.400,A 0.000,B 0.000,C 90.000,E1 71.945} C_DIS
LIN {X -0.050,Y -326.175,Z 1548.382,A 0.000,B 0.000,C 90.000,E1 68.827} C_DIS
LIN {X 0.030,Y -310.110,Z 1548.363,A 0.000,B 0.000,C 90.000,E1 65.305} C_DIS
LIN {X 0.148,Y -300.193,Z 1548.350,A 0.000,B 0.000,C 90.000,E1 62.999} C_DIS
LIN {X -0.076,Y -288.981,Z 1548.335,A 0.000,B 0.000,C 90.000,E1 60.383} C_DIS
LIN {X 0.043,Y -280.624,Z 1548.324,A 0.000,B 0.000,C 90.000,E1 58.329} C_DIS
LIN {X -0.068,Y -269.750,Z 1548.309,A 0.000,B 0.000,C 90.000,E1 55.595} C_DIS
LIN {X -0.043,Y -260.567,Z 1548.295,A 0.000,B 0.000,C 90.000,E1 53.130} C_DIS
LIN {X -0.058,Y -249.182,Z 1548.277,A 0.000,B 0.000,C 90.000,E1 49.908} C_DIS
LIN {X -0.100,Y -238.511,Z 1548.259,A 0.000,B 0.000,C 90.000,E1 46.620} C_DIS
LIN {X 0.055,Y -228.745,Z 1548.240,A 0.000,B 0.000,C 90.000,E1 43.218} C_DIS
LIN {X 0.058,Y -220.928,Z 1548.223,A 0.000,B 0.000,C 90.000,E1 40.172} C_DIS
LIN {X 0.066,Y -213.814,Z 1548.206,A 0.000,B 0.000,C 90.000,E1 37.076} C_DIS
LIN {X -0.139,Y -207.506,Z 1548.189,A 0.000,B 0.000,C 90.000,E1 33.992} C_DIS
LIN {X -0.089,Y -201.949,Z 1548.171,A 0.000,B 0.000,C 90.000,E1 30.797} C_DIS
LIN {X -0.044,Y -197.194,Z 1548.153,A 0.000,B 0.000,C 90.000,E1 27.564} C_DIS
LIN {X 0.057,Y -192.148,Z 1548.130,A 0.000,B 0.000,C 90.000,E1 23.462} C_DIS
LIN {X -0.109,Y -187.863,Z 1548.108,A 0.000,B 0.000,C 90.000,E1 19.396} C_DIS
LIN {X 0.051,Y -183.676,Z 1548.080,A 0.000,B 0.000,C 90.000,E1 14.356} C_DIS
LIN {X -0.056,Y -180.003,Z 1548.047,A 0.000,B 0.000,C 90.000,E1 8.511} C_DIS
LIN {X 0.042,Y -177.492,Z 1548.005,A 0.000,B 0.000,C 90.000,E1 0.859} C_DIS
LIN {X -0.019,Y -178.842,Z 1547.941,A 0.000,B 0.000,C 90.000,E1 349.342} C_DIS
LIN {X -0.071,Y -181.454,Z 1547.913,A 0.000,B 0.000,C 90.000,E1 344.283} C_DIS
LIN {X -0.013,Y -184.695,Z 1547.889,A 0.000,B 0.000,C 90.000,E1 340.061} C_DIS
LIN {X 0.057,Y -188.867,Z 1547.866,A 0.000,B 0.000,C 90.000,E1 335.869} C_DIS
LIN {X -0.043,Y -194.058,Z 1547.843,A 0.000,B 0.000,C 90.000,E1 331.769} C_DIS
LIN {X 0.054,Y -200.099,Z 1547.820,A 0.000,B 0.000,C 90.000,E1 327.661} C_DIS
LIN {X -0.110,Y -205.694,Z 1547.802,A 0.000,B 0.000,C 90.000,E1 324.482} C_DIS
LIN {X 0.061,Y -212.079,Z 1547.785,A 0.000,B 0.000,C 90.000,E1 321.251} C_DIS
LIN {X -0.135,Y -219.339,Z 1547.767,A 0.000,B 0.000,C 90.000,E1 318.162} C_DIS
LIN {X -0.076,Y -228.388,Z 1547.748,A 0.000,B 0.000,C 90.000,E1 314.676} C_DIS
LIN {X -0.011,Y -237.506,Z 1547.731,A 0.000,B 0.000,C 90.000,E1 311.634} C_DIS
LIN {X -0.004,Y -243.972,Z 1547.721,A 0.000,B 0.000,C 90.000,E1 309.769} C_DIS
LIN {X -0.027,Y -249.802,Z 1547.713,A 0.000,B 0.000,C 90.000,E1 308.302} C_DIS
LIN {X -0.131,Y -256.332,Z 1547.705,A 0.000,B 0.000,C 90.000,E1 306.870} C_DIS
LIN {X 0.109,Y -265.511,Z 1547.695,A 0.000,B 0.000,C 90.000,E1 305.025} C_DIS
LIN {X -0.029,Y -275.830,Z 1547.685,A 0.000,B 0.000,C 90.000,E1 303.293} C_DIS
LIN {X 0.053,Y -289.497,Z 1547.673,A 0.000,B 0.000,C 90.000,E1 301.209} C_DIS
LIN {X -0.104,Y -309.238,Z 1547.659,A 0.000,B 0.000,C 90.000,E1 298.565} C_DIS
LIN {X -0.084,Y -324.602,Z 1547.648,A 0.000,B 0.000,C 90.000,E1 296.616} C_DIS
LIN {X 0.073,Y -342.826,Z 1547.635,A 0.000,B 0.000,C 90.000,E1 294.387} C_DIS
LIN {X 0.094,Y -361.444,Z 1547.624,A 0.000,B 0.000,C 90.000,E1 292.280} C_DIS
LIN {X -0.019,Y -374.666,Z 1547.616,A 0.000,B 0.000,C 90.000,E1 290.865} C_DIS
LIN {X -0.115,Y -384.783,Z 1547.610,A 0.000,B 0.000,C 90.000,E1 289.758} C_DIS
LIN {X -0.129,Y -392.123,Z 1547.605,A 0.000,B 0.000,C 90.000,E1 288.906} C_DIS
LIN {X -0.136,Y -398.932,Z 1547.600,A 0.000,B 0.000,C 90.000,E1 288.055} C_DIS
LIN {X -0.210,Y -405.089,Z 1547.595,A 0.000,B 0.000,C 90.000,E1 287.221} C_DIS
LIN {X -0.103,Y -410.526,Z 1547.591,A 0.000,B 0.000,C 90.000,E1 286.370} C_DIS
LIN {X -0.069,Y -415.144,Z 1547.586,A 0.000,B 0.000,C 90.000,E1 285.536} C_DIS
LIN {X -0.094,Y -418.907,Z 1547.582,A 0.000,B 0.000,C 90.000,E1 284.717} C_DIS
LIN {X 0.021,Y -421.892,Z 1547.577,A 0.000,B 0.000,C 90.000,E1 283.883} C_DIS
LIN {X -0.096,Y -423.502,Z 1547.574,A 0.000,B 0.000,C 90.000,E1 283.355} C_DIS
LIN {X -0.201,Y -424.725,Z 1547.571,A 0.000,B 0.000,C 90.000,E1 282.827} C_DIS
LIN {X 0.119,Y -425.486,Z 1547.568,A 0.000,B 0.000,C 90.000,E1 282.243} C_DIS
LIN {X 0.031,Y -425.759,Z 1547.565,A 0.000,B 0.000,C 90.000,E1 281.715} C_DIS
LIN {X -0.053,Y -425.568,Z 1547.562,A 0.000,B 0.000,C 90.000,E1 281.186} C_DIS
LIN {X -0.137,Y -424.763,Z 1547.559,A 0.000,B 0.000,C 90.000,E1 280.658} C_DIS
LIN {X 0.192,Y -423.480,Z 1547.556,A 0.000,B 0.000,C 90.000,E1 280.074} C_DIS
LIN {X 0.028,Y -421.470,Z 1547.553,A 0.000,B 0.000,C 90.000,E1 279.557} C_DIS
LIN {X -0.073,Y -418.777,Z 1547.550,A 0.000,B 0.000,C 90.000,E1 279.029} C_DIS
LIN {X 0.154,Y -415.267,Z 1547.547,A 0.000,B 0.000,C 90.000,E1 278.454} C_DIS
LIN {X -0.045,Y -410.910,Z 1547.544,A 0.000,B 0.000,C 90.000,E1 277.936} C_DIS
LIN {X 0.194,Y -405.625,Z 1547.541,A 0.000,B 0.000,C 90.000,E1 277.352} C_DIS
LIN {X 0.188,Y -399.853,Z 1547.538,A 0.000,B 0.000,C 90.000,E1 276.834} C_DIS
LIN {X 0.116,Y -393.825,Z 1547.536,A 0.000,B 0.000,C 90.000,E1 276.372} C_DIS
LIN {X -0.058,Y -387.521,Z 1547.533,A 0.000,B 0.000,C 90.000,E1 275.967} C_DIS
LIN {X 0.045,Y -381.159,Z 1547.531,A 0.000,B 0.000,C 90.000,E1 275.568} C_DIS
LIN {X 0.062,Y -374.709,Z 1547.529,A 0.000,B 0.000,C 90.000,E1 275.220} C_DIS
LIN {X 0.065,Y -365.050,Z 1547.526,A 0.000,B 0.000,C 90.000,E1 274.759} C_DIS
LIN {X 0.157,Y -352.236,Z 1547.523,A 0.000,B 0.000,C 90.000,E1 274.188} C_DIS
LIN {X -0.123,Y -342.689,Z 1547.521,A 0.000,B 0.000,C 90.000,E1 273.841} C_DIS
LIN {X 0.102,Y -332.790,Z 1547.519,A 0.000,B 0.000,C 90.000,E1 273.440} C_DIS
LIN {X -0.103,Y -322.840,Z 1547.517,A 0.000,B 0.000,C 90.000,E1 273.151} C_DIS
LIN {X 0.003,Y -309.155,Z 1547.515,A 0.000,B 0.000,C 90.000,E1 272.751} C_DIS
LIN {X -0.055,Y -298.510,Z 1547.514,A 0.000,B 0.000,C 90.000,E1 272.522} C_DIS
LIN {X 0.087,Y -286.295,Z 1547.513,A 0.000,B 0.000,C 90.000,E1 272.293} C_DIS
LIN {X 0.098,Y -276.774,Z 1547.512,A 0.000,B 0.000,C 90.000,E1 272.178} C_DIS
LIN {X -0.100,Y -263.716,Z 1547.512,A 0.000,B 0.000,C 90.000,E1 272.121} C_DIS
LIN {X 0.067,Y -259.353,Z 1547.512,A 0.000,B 0.000,C 90.000,E1 272.064} C_DIS
LIN {X 0.014,Y -181.251,Z 1547.511,A 0.000,B 0.000,C 90.000,E1 272.064} C_DIS
LIN {X -0.038,Y -181.580,Z 1547.502,A 0.000,B 0.000,C 90.000,E1 270.344} C_DIS
LIN {X -0.062,Y -180.903,Z 1547.474,A 0.000,B 0.000,C 90.000,E1 265.298} C_DIS
LIN {X 0.068,Y -180.235,Z 1547.464,A 0.000,B 0.000,C 90.000,E1 263.571} C_DIS
LIN {X -0.093,Y -178.719,Z 1547.441,A 0.000,B 0.000,C 90.000,E1 259.398} C_DIS
LIN {X -0.024,Y -175.767,Z 1547.413,A 0.000,B 0.000,C 90.000,E1 254.283} C_DIS
LIN {X 0.025,Y -171.951,Z 1547.384,A 0.000,B 0.000,C 90.000,E1 249.135} C_DIS
LIN {X 0.001,Y -171.340,Z 1547.379,A 0.000,B 0.000,C 90.000,E1 248.284} C_DIS
LIN {X -0.021,Y -167.593,Z 1547.355,A 0.000,B 0.000,C 90.000,E1 243.973} C_DIS
LIN {X -0.008,Y -166.233,Z 1547.346,A 0.000,B 0.000,C 90.000,E1 242.231} C_DIS
LIN {X -0.019,Y -162.992,Z 1547.326,A 0.000,B 0.000,C 90.000,E1 238.742} C_DIS
LIN {X 0.028,Y -160.910,Z 1547.312,A 0.000,B 0.000,C 90.000,E1 236.087} C_DIS
LIN {X 0.005,Y -157.675,Z 1547.292,A 0.000,B 0.000,C 90.000,E1 232.557} C_DIS
LIN {X -0.057,Y -155.714,Z 1547.277,A 0.000,B 0.000,C 90.000,E1 229.908} C_DIS
LIN {X -0.003,Y -151.975,Z 1547.252,A 0.000,B 0.000,C 90.000,E1 225.405} C_DIS
LIN {X 0.014,Y -150.218,Z 1547.237,A 0.000,B 0.000,C 90.000,E1 222.690} C_DIS
LIN {X -0.062,Y -146.983,Z 1547.212,A 0.000,B 0.000,C 90.000,E1 218.177} C_DIS
LIN {X 0.047,Y -145.569,Z 1547.197,A 0.000,B 0.000,C 90.000,E1 215.391} C_DIS
LIN {X 0.046,Y -142.959,Z 1547.171,A 0.000,B 0.000,C 90.000,E1 210.797} C_DIS
LIN {X -0.023,Y -141.585,Z 1547.151,A 0.000,B 0.000,C 90.000,E1 207.129} C_DIS
LIN {X 0.023,Y -139.418,Z 1547.115,A 0.000,B 0.000,C 90.000,E1 200.610} C_DIS
LIN {X -0.056,Y -139.143,Z 1547.104,A 0.000,B 0.000,C 90.000,E1 198.779} C_DIS
LIN {X -0.034,Y -138.347,Z 1547.057,A 0.000,B 0.000,C 90.000,E1 190.366} C_DIS
LIN {X -0.048,Y -139.490,Z 1547.006,A 0.000,B 0.000,C 90.000,E1 181.031} C_DIS
LIN {X 0.033,Y -141.097,Z 1546.975,A 0.000,B 0.000,C 90.000,E1 175.412} C_DIS
LIN {X -0.014,Y -142.476,Z 1546.959,A 0.000,B 0.000,C 90.000,E1 172.648} C_DIS
LIN {X 0.075,Y -144.724,Z 1546.933,A 0.000,B 0.000,C 90.000,E1 167.993} C_DIS
LIN {X 0.026,Y -147.326,Z 1546.913,A 0.000,B 0.000,C 90.000,E1 164.338} C_DIS
LIN {X 0.091,Y -150.648,Z 1546.888,A 0.000,B 0.000,C 90.000,E1 159.752} C_DIS
LIN {X -0.027,Y -154.127,Z 1546.868,A 0.000,B 0.000,C 90.000,E1 156.177} C_DIS
LIN {X 0.035,Y -157.553,Z 1546.848,A 0.000,B 0.000,C 90.000,E1 152.564} C_DIS
LIN {X 0.061,Y -161.794,Z 1546.828,A 0.000,B 0.000,C 90.000,E1 148.997} C_DIS
LIN {X -0.057,Y -165.986,Z 1546.808,A 0.000,B 0.000,C 90.000,E1 145.515} C_DIS
LIN {X 0.074,Y -170.983,Z 1546.789,A 0.000,B 0.000,C 90.000,E1 141.984} C_DIS
LIN {X -0.010,Y -175.852,Z 1546.770,A 0.000,B 0.000,C 90.000,E1 138.566} C_DIS
LIN {X -0.016,Y -181.458,Z 1546.751,A 0.000,B 0.000,C 90.000,E1 135.162} C_DIS
LIN {X 0.121,Y -186.967,Z 1546.732,A 0.000,B 0.000,C 90.000,E1 131.757} C_DIS
LIN {X -0.022,Y -190.082,Z 1546.723,A 0.000,B 0.000,C 90.000,E1 130.135} C_DIS
LIN {X 0.027,Y -195.855,Z 1546.705,A 0.000,B 0.000,C 90.000,E1 126.824} C_DIS
LIN {X -0.064,Y -200.687,Z 1546.691,A 0.000,B 0.000,C 90.000,E1 124.405} C_DIS
LIN {X -0.004,Y -203.184,Z 1546.683,A 0.000,B 0.000,C 90.000,E1 122.959} C_DIS
LIN {X -0.041,Y -318.937,Z 1546.683,A 0.000,B 0.000,C 90.000,E1 122.959} C_DIS
LIN {X 0.108,Y -324.245,Z 1546.682,A 0.000,B 0.000,C 90.000,E1 122.752} C_DIS
LIN {X -0.070,Y -327.391,Z 1546.681,A 0.000,B 0.000,C 90.000,E1 122.546} C_DIS
LIN {X 0.027,Y -331.094,Z 1546.678,A 0.000,B 0.000,C 90.000,E1 122.084} C_DIS
LIN {X -0.147,Y -332.927,Z 1546.677,A 0.000,B 0.000,C 90.000,E1 121.799} C_DIS
LIN {X 0.089,Y -335.547,Z 1546.673,A 0.000,B 0.000,C 90.000,E1 121.131} C_DIS
LIN {X 0.018,Y -347.007,Z 1546.658,A 0.000,B 0.000,C 90.000,E1 118.359} C_DIS
LIN {X -0.062,Y -359.878,Z 1546.642,A 0.000,B 0.000,C 90.000,E1 115.643} C_DIS
LIN {X 0.079,Y -374.278,Z 1546.628,A 0.000,B 0.000,C 90.000,E1 112.950} C_DIS
LIN {X -0.150,Y -388.458,Z 1546.615,A 0.000,B 0.000,C 90.000,E1 110.663} C_DIS
LIN {X 0.068,Y -404.039,Z 1546.602,A 0.000,B 0.000,C 90.000,E1 108.362} C_DIS
LIN {X 0.056,Y -421.130,Z 1546.590,A 0.000,B 0.000,C 90.000,E1 106.150} C_DIS
LIN {X -0.063,Y -439.850,Z 1546.578,A 0.000,B 0.000,C 90.000,E1 104.008} C_DIS
LIN {X 0.047,Y -459.765,Z 1546.566,A 0.000,B 0.000,C 90.000,E1 101.951} C_DIS
LIN {X 0.061,Y -482.819,Z 1546.555,A 0.000,B 0.000,C 90.000,E1 99.849} C_DIS
LIN {X 0.090,Y -493.108,Z 1546.550,A 0.000,B 0.000,C 90.000,E1 98.973} C_DIS
LIN {X 0.200,Y -494.978,Z 1546.549,A 0.000,B 0.000,C 90.000,E1 98.746} C_DIS
LIN {X 0.114,Y -496.606,Z 1546.547,A 0.000,B 0.000,C 90.000,E1 98.511} C_DIS
LIN {X 0.024,Y -497.820,Z 1546.546,A 0.000,B 0.000,C 90.000,E1 98.276} C_DIS
LIN {X -0.208,Y -499.283,Z 1546.543,A 0.000,B 0.000,C 90.000,E1 97.814} C_DIS
LIN {X 0.062,Y -499.681,Z 1546.541,A 0.000,B 0.000,C 90.000,E1 97.296} C_DIS
LIN {X -0.154,Y -499.081,Z 1546.538,A 0.000,B 0.000,C 90.000,E1 96.834} C_DIS
LIN {X 0.128,Y -497.389,Z 1546.535,A 0.000,B 0.000,C 90.000,E1 96.315} C_DIS
LIN {X -0.007,Y -496.036,Z 1546.534,A 0.000,B 0.000,C 90.000,E1 96.087} C_DIS
LIN {X -0.069,Y -483.159,Z 1546.523,A 0.000,B 0.000,C 90.000,E1 94.131} C_DIS
LIN {X 0.105,Y -475.312,Z 1546.516,A 0.000,B 0.000,C 90.000,E1 92.865} C_DIS
LIN {X 0.129,Y -467.056,Z 1546.509,A 0.000,B 0.000,C 90.000,E1 91.604} C_DIS
LIN {X 0.030,Y -458.422,Z 1546.502,A 0.000,B 0.000,C 90.000,E1 90.344} C_DIS
LIN {X -0.191,Y -449.496,Z 1546.495,A 0.000,B 0.000,C 90.000,E1 89.083} C_DIS
LIN {X -0.073,Y -440.153,Z 1546.488,A 0.000,B 0.000,C 90.000,E1 87.764} C_DIS
LIN {X 0.051,Y -428.654,Z 1546.479,A 0.000,B 0.000,C 90.000,E1 86.159} C_DIS
LIN {X 0.124,Y -415.100,Z 1546.468,A 0.000,B 0.000,C 90.000,E1 84.261} C_DIS
LIN {X 0.066,Y -400.079,Z 1546.456,A 0.000,B 0.000,C 90.000,E1 82.064} C_DIS
LIN {X -0.139,Y -380.513,Z 1546.439,A 0.000,B 0.000,C 90.000,E1 78.982} C_DIS
LIN {X -0.075,Y -363.842,Z 1546.422,A 0.000,B 0.000,C 90.000,E1 76.061} C_DIS
LIN {X -0.133,Y -350.934,Z 1546.409,A 0.000,B 0.000,C 90.000,E1 73.685} C_DIS
LIN {X 0.128,Y -341.320,Z 1546.399,A 0.000,B 0.000,C 90.000,E1 71.819} C_DIS
LIN {X 0.095,Y -325.803,Z 1546.382,A 0.000,B 0.000,C 90.000,E1 68.720} C_DIS
LIN {X -0.010,Y -309.750,Z 1546.362,A 0.000,B 0.000,C 90.000,E1 65.229} C_DIS
LIN {X -0.030,Y -299.836,Z 1546.350,A 0.000,B 0.000,C 90.000,E1 62.948} C_DIS
LIN {X 0.133,Y -288.637,Z 1546.335,A 0.000,B 0.000,C 90.000,E1 60.255} C_DIS
LIN {X -0.041,Y -278.928,Z 1546.322,A 0.000,B 0.000,C 90.000,E1 57.916} C_DIS
LIN {X 0.032,Y -268.121,Z 1546.306,A 0.000,B 0.000,C 90.000,E1 55.135} C_DIS
LIN {X 0.012,Y -257.709,Z 1546.291,A 0.000,B 0.000,C 90.000,E1 52.316} C_DIS
LIN {X -0.082,Y -246.522,Z 1546.273,A 0.000,B 0.000,C 90.000,E1 49.094} C_DIS
LIN {X 0.123,Y -236.088,Z 1546.254,A 0.000,B 0.000,C 90.000,E1 45.729} C_DIS
LIN {X 0.054,Y -226.622,Z 1546.235,A 0.000,B 0.000,C 90.000,E1 42.366} C_DIS
LIN {X 0.003,Y -219.044,Z 1546.219,A 0.000,B 0.000,C 90.000,E1 39.322} C_DIS
LIN {X 0.000,Y -212.186,Z 1546.201,A 0.000,B 0.000,C 90.000,E1 36.217} C_DIS
LIN {X -0.073,Y -206.111,Z 1546.184,A 0.000,B 0.000,C 90.000,E1 33.086} C_DIS
LIN {X 0.005,Y -200.804,Z 1546.166,A 0.000,B 0.000,C 90.000,E1 29.873} C_DIS
LIN {X -0.048,Y -195.228,Z 1546.144,A 0.000,B 0.000,C 90.000,E1 25.848} C_DIS
LIN {X 0.093,Y -190.517,Z 1546.121,A 0.000,B 0.000,C 90.000,E1 21.716} C_DIS
LIN {X -0.081,Y -186.533,Z 1546.098,A 0.000,B 0.000,C 90.000,E1 17.638} C_DIS
LIN {X 0.055,Y -182.688,Z 1546.070,A 0.000,B 0.000,C 90.000,E1 12.591} C_DIS
LIN {X -0.007,Y -179.436,Z 1546.037,A 0.000,B 0.000,C 90.000,E1 6.720} C_DIS
LIN {X 0.033,Y -177.459,Z 1545.988,A 0.000,B 0.000,C 90.000,E1 357.822} C_DIS
LIN {X 0.001,Y -179.094,Z 1545.941,A 0.000,B 0.000,C 90.000,E1 349.342} C_DIS
LIN {X -0.015,Y -182.284,Z 1545.908,A 0.000,B 0.000,C 90.000,E1 343.433} C_DIS
LIN {X 0.075,Y -185.682,Z 1545.885,A 0.000,B 0.000,C 90.000,E1 339.209} C_DIS
LIN {X -0.099,Y -190.039,Z 1545.861,A 0.000,B 0.000,C 90.000,E1 335.101} C_DIS
LIN {X 0.101,Y -195.381,Z 1545.839,A 0.000,B 0.000,C 90.000,E1 330.923} C_DIS
LIN {X -0.053,Y -200.277,Z 1545.821,A 0.000,B 0.000,C 90.000,E1 327.709} C_DIS
LIN {X -0.042,Y -205.826,Z 1545.803,A 0.000,B 0.000,C 90.000,E1 324.482} C_DIS
LIN {X -0.031,Y -212.193,Z 1545.785,A 0.000,B 0.000,C 90.000,E1 321.295} C_DIS
LIN {X -0.055,Y -219.425,Z 1545.767,A 0.000,B 0.000,C 90.000,E1 318.162} C_DIS
LIN {X 0.003,Y -228.453,Z 1545.748,A 0.000,B 0.000,C 90.000,E1 314.676} C_DIS
LIN {X -0.106,Y -237.516,Z 1545.731,A 0.000,B 0.000,C 90.000,E1 311.676} C_DIS
LIN {X -0.074,Y -243.972,Z 1545.721,A 0.000,B 0.000,C 90.000,E1 309.806} C_DIS
LIN {X 0.060,Y -249.776,Z 1545.713,A 0.000,B 0.000,C 90.000,E1 308.302} C_DIS
LIN {X -0.042,Y -256.248,Z 1545.705,A 0.000,B 0.000,C 90.000,E1 306.870} C_DIS
LIN {X -0.065,Y -263.477,Z 1545.697,A 0.000,B 0.000,C 90.000,E1 305.438} C_DIS
LIN {X -0.008,Y -273.525,Z 1545.687,A 0.000,B 0.000,C 90.000,E1 303.658} C_DIS
LIN {X -0.061,Y -286.931,Z 1545.675,A 0.000,B 0.000,C 90.000,E1 301.592} C_DIS
LIN {X -0.009,Y -309.050,Z 1545.659,A 0.000,B 0.000,C 90.000,E1 298.565} C_DIS
LIN {X 0.013,Y -324.460,Z 1545.648,A 0.000,B 0.000,C 90.000,E1 296.616} C_DIS
LIN {X -0.177,Y -342.622,Z 1545.636,A 0.000,B 0.000,C 90.000,E1 294.463} C_DIS
LIN {X 0.020,Y -361.246,Z 1545.624,A 0.000,B 0.000,C 90.000,E1 292.333} C_DIS
LIN {X 0.018,Y -374.348,Z 1545.616,A 0.000,B 0.000,C 90.000,E1 290.918} C_DIS
LIN {X 0.098,Y -381.988,Z 1545.612,A 0.000,B 0.000,C 90.000,E1 290.066} C_DIS
LIN {X 0.021,Y -389.586,Z 1545.607,A 0.000,B 0.000,C 90.000,E1 289.214} C_DIS
LIN {X -0.010,Y -396.641,Z 1545.602,A 0.000,B 0.000,C 90.000,E1 288.362} C_DIS
LIN {X 0.026,Y -403.081,Z 1545.597,A 0.000,B 0.000,C 90.000,E1 287.511} C_DIS
LIN {X -0.008,Y -408.798,Z 1545.593,A 0.000,B 0.000,C 90.000,E1 286.677} C_DIS
LIN {X 0.020,Y -413.782,Z 1545.588,A 0.000,B 0.000,C 90.000,E1 285.843} C_DIS
LIN {X 0.088,Y -417.855,Z 1545.583,A 0.000,B 0.000,C 90.000,E1 285.009} C_DIS
LIN {X -0.049,Y -420.134,Z 1545.580,A 0.000,B 0.000,C 90.000,E1 284.481} C_DIS
LIN {X -0.069,Y -422.117,Z 1545.577,A 0.000,B 0.000,C 90.000,E1 283.939} C_DIS
LIN {X -0.187,Y -423.741,Z 1545.574,A 0.000,B 0.000,C 90.000,E1 283.411} C_DIS
LIN {X 0.122,Y -425.027,Z 1545.571,A 0.000,B 0.000,C 90.000,E1 282.827} C_DIS
LIN {X 0.029,Y -425.861,Z 1545.568,A 0.000,B 0.000,C 90.000,E1 282.299} C_DIS
LIN {X -0.059,Y -426.225,Z 1545.565,A 0.000,B 0.000,C 90.000,E1 281.771} C_DIS
LIN {X -0.141,Y -426.085,Z 1545.562,A 0.000,B 0.000,C 90.000,E1 281.243} C_DIS
LIN {X 0.195,Y -425.401,Z 1545.559,A 0.000,B 0.000,C 90.000,E1 280.658} C_DIS
LIN {X 0.035,Y -424.150,Z 1545.556,A 0.000,B 0.000,C 90.000,E1 280.141} C_DIS
LIN {X -0.052,Y -422.269,Z 1545.553,A 0.000,B 0.000,C 90.000,E1 279.613} C_DIS
LIN {X -0.149,Y -419.692,Z 1545.550,A 0.000,B 0.000,C 90.000,E1 279.086} C_DIS
LIN {X 0.084,Y -416.305,Z 1545.547,A 0.000,B 0.000,C 90.000,E1 278.511} C_DIS
LIN {X -0.111,Y -411.970,Z 1545.544,A 0.000,B 0.000,C 90.000,E1 277.992} C_DIS
LIN {X 0.136,Y -406.856,Z 1545.541,A 0.000,B 0.000,C 90.000,E1 277.409} C_DIS
LIN {X 0.058,Y -400.992,Z 1545.538,A 0.000,B 0.000,C 90.000,E1 276.891} C_DIS
LIN {X -0.051,Y -394.936,Z 1545.536,A 0.000,B 0.000,C 90.000,E1 276.429} C_DIS
LIN {X 0.161,Y -388.637,Z 1545.533,A 0.000,B 0.000,C 90.000,E1 275.967} C_DIS
LIN {X -0.090,Y -382.445,Z 1545.531,A 0.000,B 0.000,C 90.000,E1 275.625} C_DIS
LIN {X -0.106,Y -375.943,Z 1545.529,A 0.000,B 0.000,C 90.000,E1 275.277} C_DIS
LIN {X -0.148,Y -366.232,Z 1545.527,A 0.000,B 0.000,C 90.000,E1 274.821} C_DIS
LIN {X -0.010,Y -353.512,Z 1545.524,A 0.000,B 0.000,C 90.000,E1 274.245} C_DIS
LIN {X -0.002,Y -340.796,Z 1545.521,A 0.000,B 0.000,C 90.000,E1 273.726} C_DIS
LIN {X -0.084,Y -330.619,Z 1545.519,A 0.000,B 0.000,C 90.000,E1 273.383} C_DIS
LIN {X -0.108,Y -317.412,Z 1545.516,A 0.000,B 0.000,C 90.000,E1 272.980} C_DIS
LIN {X -0.025,Y -307.032,Z 1545.515,A 0.000,B 0.000,C 90.000,E1 272.694} C_DIS
LIN {X -0.050,Y -295.861,Z 1545.514,A 0.000,B 0.000,C 90.000,E1 272.465} C_DIS
LIN {X -0.127,Y -283.399,Z 1545.513,A 0.000,B 0.000,C 90.000,E1 272.293} C_DIS
LIN {X 0.070,Y -269.503,Z 1545.512,A 0.000,B 0.000,C 90.000,E1 272.121} C_DIS
LIN {X 0.075,Y -259.174,Z 1545.512,A 0.000,B 0.000,C 90.000,E1 272.064} C_DIS
LIN {X 0.020,Y -181.250,Z 1545.511,A 0.000,B 0.000,C 90.000,E1 272.064} C_DIS
LIN {X 0.001,Y -181.579,Z 1545.502,A 0.000,B 0.000,C 90.000,E1 270.344} C_DIS
LIN {X -0.023,Y -180.904,Z 1545.474,A 0.000,B 0.000,C 90.000,E1 265.298} C_DIS
LIN {X -0.073,Y -180.241,Z 1545.464,A 0.000,B 0.000,C 90.000,E1 263.628} C_DIS
LIN {X -0.054,Y -178.726,Z 1545.441,A 0.000,B 0.000,C 90.000,E1 259.398} C_DIS
LIN {X 0.013,Y -175.775,Z 1545.413,A 0.000,B 0.000,C 90.000,E1 254.283} C_DIS
LIN {X 0.002,Y -171.958,Z 1545.384,A 0.000,B 0.000,C 90.000,E1 249.156} C_DIS
LIN {X 0.039,Y -171.352,Z 1545.379,A 0.000,B 0.000,C 90.000,E1 248.284} C_DIS
LIN {X 0.016,Y -167.602,Z 1545.355,A 0.000,B 0.000,C 90.000,E1 243.973} C_DIS
LIN {X 0.029,Y -166.246,Z 1545.346,A 0.000,B 0.000,C 90.000,E1 242.231} C_DIS
LIN {X 0.016,Y -163.003,Z 1545.326,A 0.000,B 0.000,C 90.000,E1 238.742} C_DIS
LIN {X 0.063,Y -160.923,Z 1545.312,A 0.000,B 0.000,C 90.000,E1 236.087} C_DIS
LIN {X 0.041,Y -157.686,Z 1545.292,A 0.000,B 0.000,C 90.000,E1 232.557} C_DIS
LIN {X -0.021,Y -155.725,Z 1545.277,A 0.000,B 0.000,C 90.000,E1 229.908} C_DIS
LIN {X 0.033,Y -151.984,Z 1545.252,A 0.000,B 0.000,C 90.000,E1 225.405} C_DIS
LIN {X 0.048,Y -150.228,Z 1545.237,A 0.000,B 0.000,C 90.000,E1 222.690} C_DIS
LIN {X -0.028,Y -146.991,Z 1545.212,A 0.000,B 0.000,C 90.000,E1 218.177} C_DIS
LIN {X -0.038,Y -145.576,Z 1545.197,A 0.000,B 0.000,C 90.000,E1 215.438} C_DIS
LIN {X 0.079,Y -142.965,Z 1545.171,A 0.000,B 0.000,C 90.000,E1 210.797} C_DIS
LIN {X 0.010,Y -141.592,Z 1545.151,A 0.000,B 0.000,C 90.000,E1 207.129} C_DIS
LIN {X 0.057,Y -139.420,Z 1545.115,A 0.000,B 0.000,C 90.000,E1 200.610} C_DIS
LIN {X -0.022,Y -139.147,Z 1545.104,A 0.000,B 0.000,C 90.000,E1 198.779} C_DIS
LIN {X 0.000,Y -138.346,Z 1545.058,A 0.000,B 0.000,C 90.000,E1 190.366} C_DIS
LIN {X -0.015,Y -139.488,Z 1545.006,A 0.000,B 0.000,C 90.000,E1 181.031} C_DIS
LIN {X 0.065,Y -141.092,Z 1544.975,A 0.000,B 0.000,C 90.000,E1 175.412} C_DIS
LIN {X 0.019,Y -142.470,Z 1544.959,A 0.000,B 0.000,C 90.000,E1 172.648} C_DIS
LIN {X -0.032,Y -144.716,Z 1544.934,A 0.000,B 0.000,C 90.000,E1 168.049} C_DIS
LIN {X 0.060,Y -147.316,Z 1544.913,A 0.000,B 0.000,C 90.000,E1 164.338} C_DIS
LIN {X -0.015,Y -150.638,Z 1544.888,A 0.000,B 0.000,C 90.000,E1 159.806} C_DIS
LIN {X 0.008,Y -154.114,Z 1544.868,A 0.000,B 0.000,C 90.000,E1 156.177} C_DIS
